IF VI_Sensor_Fault THEN
    L_Sensor_Fault_Clear_Count := 0;
    IF L_Sensor_Fault_Assert_Count < C_HEALTH_DEBOUNCE_CYCLES THEN
        L_Sensor_Fault_Assert_Count := L_Sensor_Fault_Assert_Count + 1;
    END_IF;
    IF L_Sensor_Fault_Assert_Count >= C_HEALTH_DEBOUNCE_CYCLES THEN
        L_Sensor_Fault_Stable := TRUE;
    END_IF;
ELSE
    L_Sensor_Fault_Assert_Count := 0;
    IF L_Sensor_Fault_Clear_Count < C_HEALTH_DEBOUNCE_CYCLES THEN
        L_Sensor_Fault_Clear_Count := L_Sensor_Fault_Clear_Count + 1;
    END_IF;
    IF L_Sensor_Fault_Clear_Count >= C_HEALTH_DEBOUNCE_CYCLES THEN
        L_Sensor_Fault_Stable := FALSE;
    END_IF;
END_IF;

IF VI_Subsystem_Fault THEN
    L_Subsystem_Clear_Count := 0;
    IF L_Subsystem_Assert_Count < C_HEALTH_DEBOUNCE_CYCLES THEN
        L_Subsystem_Assert_Count := L_Subsystem_Assert_Count + 1;
    END_IF;
    IF L_Subsystem_Assert_Count >= C_HEALTH_DEBOUNCE_CYCLES THEN
        L_Subsystem_Fault_Stable := TRUE;
    END_IF;
ELSE
    L_Subsystem_Assert_Count := 0;
    IF L_Subsystem_Clear_Count < C_HEALTH_DEBOUNCE_CYCLES THEN
        L_Subsystem_Clear_Count := L_Subsystem_Clear_Count + 1;
    END_IF;
    IF L_Subsystem_Clear_Count >= C_HEALTH_DEBOUNCE_CYCLES THEN
        L_Subsystem_Fault_Stable := FALSE;
    END_IF;
END_IF;

// Count confirmed fault events on rising edge of stable/critical conditions
IF L_IO_Fault_Stable AND NOT L_IO_Fault_Prev THEN
    VO_IO_Fault_Count := VO_IO_Fault_Count + 1;
END_IF;
L_IO_Fault_Prev := L_IO_Fault_Stable;

IF L_Comm_Fault_Stable AND NOT L_Comm_Fault_Prev THEN
    VO_Comm_Fault_Count := VO_Comm_Fault_Count + 1;
END_IF;
L_Comm_Fault_Prev := L_Comm_Fault_Stable;

IF L_Sensor_Fault_Stable AND NOT L_Sensor_Fault_Prev THEN
    VO_Sensor_Fault_Count := VO_Sensor_Fault_Count + 1;
END_IF;
L_Sensor_Fault_Prev := L_Sensor_Fault_Stable;

IF L_Subsystem_Fault_Stable AND NOT L_Subsystem_Fault_Prev THEN
    VO_Subsystem_Fault_Count := VO_Subsystem_Fault_Count + 1;
END_IF;
L_Subsystem_Fault_Prev := L_Subsystem_Fault_Stable;

IF VI_Watchdog_Fault AND NOT L_Watchdog_Fault_Prev THEN
    VO_Watchdog_Fault_Count := VO_Watchdog_Fault_Count + 1;
END_IF;
L_Watchdog_Fault_Prev := VI_Watchdog_Fault;

VO_Sensor_Fault := L_Sensor_Fault_Stable;
VO_IO_Fault := L_IO_Fault_Stable;
VO_Comm_Fault := L_Comm_Fault_Stable;
VO_Subsystem_Degraded := L_Subsystem_Fault_Stable;

VO_System_Severity := E_System_Severity.SEV_NORMAL;
VO_Root_Cause := E_System_Root_Cause.ROOT_NONE;
VO_First_Fault_Active := FALSE;
VO_First_Fault_Type := 0;
VO_First_Fault_Source := 0;

// Priority: FIRE > GAS > CO > WATER > diagnostics
IF VI_Smoke_Detected THEN
    VO_System_Severity := E_System_Severity.SEV_CRITICAL;
    VO_Root_Cause := E_System_Root_Cause.ROOT_FIRE;
    VO_First_Fault_Active := TRUE;
    VO_First_Fault_Type := 5;

ELSIF VI_Gas_Detected THEN
    VO_System_Severity := E_System_Severity.SEV_CRITICAL;
    VO_Root_Cause := E_System_Root_Cause.ROOT_GAS_LEAK;
    VO_First_Fault_Active := TRUE;
    VO_First_Fault_Type := 6;

ELSIF VI_CO_Alarm_Level THEN
    VO_System_Severity := E_System_Severity.SEV_CRITICAL;
    VO_Root_Cause := E_System_Root_Cause.ROOT_CO_CRITICAL;
    VO_First_Fault_Active := TRUE;
    VO_First_Fault_Type := 7;

ELSIF VI_CO_Warning_Level THEN
    VO_System_Severity := E_System_Severity.SEV_WARNING;
    VO_Root_Cause := E_System_Root_Cause.ROOT_CO_WARNING;
    VO_First_Fault_Active := TRUE;
    VO_First_Fault_Type := 7;

ELSIF VI_Leak_Detected THEN
    VO_System_Severity := E_System_Severity.SEV_WARNING;
    VO_Root_Cause := E_System_Root_Cause.ROOT_WATER_LEAK;
    VO_First_Fault_Active := TRUE;
    VO_First_Fault_Type := 8;

ELSIF VI_Watchdog_Fault THEN
    VO_System_Severity := E_System_Severity.SEV_CRITICAL;
    VO_Root_Cause := E_System_Root_Cause.ROOT_WATCHDOG_FAULT;
    VO_First_Fault_Active := TRUE;
    VO_First_Fault_Type := 9;

ELSIF L_IO_Fault_Stable THEN
    VO_System_Severity := E_System_Severity.SEV_DEGRADED;
    VO_Root_Cause := E_System_Root_Cause.ROOT_IO_OFFLINE;
    VO_First_Fault_Active := TRUE;
    VO_First_Fault_Type := 1;

ELSIF L_Comm_Fault_Stable THEN
    VO_System_Severity := E_System_Severity.SEV_DEGRADED;
    VO_Root_Cause := E_System_Root_Cause.ROOT_COMM_FAULT;
    VO_First_Fault_Active := TRUE;
    VO_First_Fault_Type := 3;

ELSIF L_Sensor_Fault_Stable THEN
    VO_System_Severity := E_System_Severity.SEV_DEGRADED;
    VO_Root_Cause := E_System_Root_Cause.ROOT_SENSOR_FAULT;
    VO_First_Fault_Active := TRUE;
    VO_First_Fault_Type := 2;

ELSIF L_Subsystem_Fault_Stable THEN
    VO_System_Severity := E_System_Severity.SEV_DEGRADED;
    VO_Root_Cause := E_System_Root_Cause.ROOT_SUBSYSTEM_FAULT;
    VO_First_Fault_Active := TRUE;
    VO_First_Fault_Type := 4;
END_IF;
// >>> BULK_SYNC_ANCHOR: FB_System_Health <<<
          
END_FUNCTION_BLOCK

FUNCTION_BLOCK FB_Rule_Engine
  VAR_INPUT
    VI_System_Time_MS : UDINT;
    VI_IsActivePLC : BOOL;
    VI_Security_Armed : BOOL;
    VI_Current_Time : TOD;
    VI_Day_Of_Week : INT;
  END_VAR
  VAR_OUTPUT
    VO_Preheat_Request : BOOL;
    VO_Actions : ARRAY[1..GVL_CONSTANTS.C_MAX_RULES] OF ST_Rule_Action;
  END_VAR
  VAR_IN_OUT
    VI_Rules : ARRAY[1..GVL_CONSTANTS.C_MAX_RULES] OF ST_User_Rule;
    VI_Indoor_Temps : ARRAY[1..16] OF REAL;
    VI_Floor_Temps : ARRAY[1..GVL_CONSTANTS.C_MAX_HEATING_CIRCUITS] OF REAL;
    VI_Humidities : ARRAY[1..16] OF REAL;
    VI_CO2_Levels : ARRAY[1..16] OF REAL;
    VI_Motion_Sensors : ARRAY[1..16] OF BOOL;
    VI_Door_Sensors : ARRAY[1..GVL_CONSTANTS.C_MAX_DOOR_SENSORS] OF BOOL;
    VI_Window_Sensors : ARRAY[1..16] OF BOOL;
    VI_Water_Sensors : ARRAY[1..GVL_CONSTANTS.C_MAX_FLOOD_SENSORS] OF BOOL;
    VI_Smoke_Sensors : ARRAY[1..GVL_CONSTANTS.C_MAX_SMOKE_SENSORS] OF BOOL;
    VI_Methane_Sensors : ARRAY[1..GVL_CONSTANTS.C_MAX_METHANE_SENSORS] OF REAL;
    VI_CO_Sensors : ARRAY[1..GVL_CONSTANTS.C_MAX_CO_SENSORS] OF REAL;
  END_VAR
  VAR
    L_i : INT;
    L_Condition_Met : BOOL;
    L_Current_Value : REAL;
    L_Triggers : ARRAY[1..GVL_CONSTANTS.C_MAX_RULES] OF R_TRIG;
    L_Trigger_Count : ARRAY[1..GVL_CONSTANTS.C_MAX_RULES] OF UINT;
    L_Last_Reset_Time : UDINT;
    L_Elapsed_Time : UDINT;
  END_VAR

            IF NOT VI_IsActivePLC THEN
    FOR L_i := 1 TO GVL_CONSTANTS.C_MAX_RULES DO
        VO_Actions[L_i].Active := FALSE;
        VO_Actions[L_i].Triggered := FALSE;
        VO_Actions[L_i].Action_Type := E_Rule_Action_Type.ACTION_NONE;
        VO_Actions[L_i].Target_ID := 0;
        VO_Actions[L_i].Value := 0.0;
    END_FOR;
    VO_Preheat_Request := FALSE;
    RETURN;
END_IF;

VO_Preheat_Request := FALSE;

L_Elapsed_Time := SEL(VI_System_Time_MS >= L_Last_Reset_Time, VI_System_Time_MS - L_Last_Reset_Time, (4294967295 - L_Last_Reset_Time) + VI_System_Time_MS + 1);

IF L_Elapsed_Time >= GVL_CONSTANTS.C_MS_IN_MINUTE THEN
    L_Last_Reset_Time := VI_System_Time_MS;
    FOR L_i := 1 TO GVL_CONSTANTS.C_MAX_RULES DO
        L_Trigger_Count[L_i] := 0;
    END_FOR;
END_IF;

FOR L_i := 1 TO GVL_CONSTANTS.C_MAX_RULES DO

    // Full per-cycle action reset prevents stale Triggered/Action_Type/Target_ID/Value
    // from being observed by any downstream consumer when a rule is disabled or inactive.
    VO_Actions[L_i].Active := FALSE;
    VO_Actions[L_i].Triggered := FALSE;
    VO_Actions[L_i].Action_Type := E_Rule_Action_Type.ACTION_NONE;
    VO_Actions[L_i].Target_ID := 0;
    VO_Actions[L_i].Value := 0.0;

    IF VI_Rules[L_i].Enabled THEN
        L_Condition_Met := FALSE;
        L_Current_Value := 0.0;
        
        IF VI_Rules[L_i].Condition_Target_ID > 0 THEN
            CASE VI_Rules[L_i].Condition_Type OF
                E_Rule_Condition_Type.COND_AIR_TEMP: IF VI_Rules[L_i].Condition_Target_ID <= 16 THEN L_Current_Value := VI_Indoor_Temps[VI_Rules[L_i].Condition_Target_ID]; END_IF;
                E_Rule_Condition_Type.COND_FLOOR_TEMP: IF VI_Rules[L_i].Condition_Target_ID <= GVL_CONSTANTS.C_MAX_HEATING_CIRCUITS THEN L_Current_Value := VI_Floor_Temps[VI_Rules[L_i].Condition_Target_ID]; END_IF;
                E_Rule_Condition_Type.COND_HUMIDITY: IF VI_Rules[L_i].Condition_Target_ID <= 16 THEN L_Current_Value := VI_Humidities[VI_Rules[L_i].Condition_Target_ID]; END_IF;
                E_Rule_Condition_Type.COND_CO2: IF VI_Rules[L_i].Condition_Target_ID <= 16 THEN L_Current_Value := VI_CO2_Levels[VI_Rules[L_i].Condition_Target_ID]; END_IF;
                E_Rule_Condition_Type.COND_MOTION: IF VI_Rules[L_i].Condition_Target_ID <= 16 THEN L_Current_Value := SEL(VI_Motion_Sensors[VI_Rules[L_i].Condition_Target_ID], 0.0, 1.0); END_IF;
                E_Rule_Condition_Type.COND_DOOR_WINDOW: 
                    IF VI_Rules[L_i].Condition_Target_ID <= GVL_CONSTANTS.C_MAX_DOOR_SENSORS THEN
                        L_Current_Value := SEL(VI_Door_Sensors[VI_Rules[L_i].Condition_Target_ID] OR VI_Window_Sensors[VI_Rules[L_i].Condition_Target_ID], 0.0, 1.0);
                    ELSIF VI_Rules[L_i].Condition_Target_ID <= 16 THEN
                        L_Current_Value := SEL(VI_Window_Sensors[VI_Rules[L_i].Condition_Target_ID], 0.0, 1.0);
                    END_IF;
                E_Rule_Condition_Type.COND_FLOOD: IF VI_Rules[L_i].Condition_Target_ID <= GVL_CONSTANTS.C_MAX_FLOOD_SENSORS THEN L_Current_Value := SEL(VI_Water_Sensors[VI_Rules[L_i].Condition_Target_ID], 0.0, 1.0); END_IF;
                E_Rule_Condition_Type.COND_SMOKE: IF VI_Rules[L_i].Condition_Target_ID <= GVL_CONSTANTS.C_MAX_SMOKE_SENSORS THEN L_Current_Value := SEL(VI_Smoke_Sensors[VI_Rules[L_i].Condition_Target_ID], 0.0, 1.0); END_IF;
                E_Rule_Condition_Type.COND_METHANE: IF VI_Rules[L_i].Condition_Target_ID <= GVL_CONSTANTS.C_MAX_METHANE_SENSORS THEN L_Current_Value := VI_Methane_Sensors[VI_Rules[L_i].Condition_Target_ID]; END_IF;
                E_Rule_Condition_Type.COND_CO: IF VI_Rules[L_i].Condition_Target_ID <= GVL_CONSTANTS.C_MAX_CO_SENSORS THEN L_Current_Value := VI_CO_Sensors[VI_Rules[L_i].Condition_Target_ID]; END_IF;
                E_Rule_Condition_Type.COND_TIME_OF_DAY: L_Current_Value := TO_REAL(TOD_TO_UDINT(VI_Current_Time) / GVL_CONSTANTS.C_MS_IN_MINUTE);
                E_Rule_Condition_Type.COND_DAY_OF_WEEK: L_Current_Value := TO_REAL(VI_Day_Of_Week);
            END_CASE;
        ELSE
            IF VI_Rules[L_i].Condition_Type = E_Rule_Condition_Type.COND_TIME_OF_DAY THEN
                L_Current_Value := TO_REAL(TOD_TO_UDINT(VI_Current_Time) / GVL_CONSTANTS.C_MS_IN_MINUTE);
            ELSIF VI_Rules[L_i].Condition_Type = E_Rule_Condition_Type.COND_DAY_OF_WEEK THEN
                L_Current_Value := TO_REAL(VI_Day_Of_Week);
            END_IF;
        END_IF;
        
        CASE VI_Rules[L_i].Condition_Op OF
            E_Rule_Comparison.COMP_GT: L_Condition_Met := (L_Current_Value > VI_Rules[L_i].Condition_Value);
            E_Rule_Comparison.COMP_LT: L_Condition_Met := (L_Current_Value < VI_Rules[L_i].Condition_Value);
            E_Rule_Comparison.COMP_EQ: L_Condition_Met := (ABS(L_Current_Value - VI_Rules[L_i].Condition_Value) < 0.1);
            E_Rule_Comparison.COMP_GE: L_Condition_Met := (L_Current_Value >= VI_Rules[L_i].Condition_Value);
            E_Rule_Comparison.COMP_LE: L_Condition_Met := (L_Current_Value <= VI_Rules[L_i].Condition_Value);
            E_Rule_Comparison.COMP_IN_RANGE: L_Condition_Met := (L_Current_Value >= VI_Rules[L_i].Condition_Value) AND (L_Current_Value <= VI_Rules[L_i].Condition_Value_Max);
            E_Rule_Comparison.COMP_TRUE: L_Condition_Met := (L_Current_Value > 0.5);
            E_Rule_Comparison.COMP_FALSE: L_Condition_Met := (L_Current_Value < 0.5);
        END_CASE;
        
        L_Triggers[L_i](CLK := L_Condition_Met);
        
        IF L_Triggers[L_i].Q THEN
            L_Trigger_Count[L_i] := L_Trigger_Count[L_i] + 1;
            IF L_Trigger_Count[L_i] > 10 THEN
                CONTINUE;
            END_IF;
        END_IF;
        
        IF L_Condition_Met AND (L_Trigger_Count[L_i] <= 10) THEN
            VO_Actions[L_i].Active := TRUE;
            VO_Actions[L_i].Triggered := L_Triggers[L_i].Q;
            VO_Actions[L_i].Action_Type := VI_Rules[L_i].Action_Type;
            VO_Actions[L_i].Target_ID := VI_Rules[L_i].Action_Target_ID;
            VO_Actions[L_i].Value := VI_Rules[L_i].Action_Value;
        END_IF;
    END_IF;
END_FOR;

// >>> BULK_SYNC_ANCHOR: FB_Rule_Engine <<<
          
END_FUNCTION_BLOCK

FUNCTION_BLOCK FB_Heating_Runtime_Service_Gating_Phase
  VAR_INPUT
    VI_Enable : BOOL;
  END_VAR
  VAR_OUTPUT
    VO_Executed : BOOL;
    VO_Valid : BOOL;
  END_VAR
  VAR_IN_OUT
    VIO_Manifold_Pumps : ARRAY[1..GVL_CONSTANTS.C_MAX_MANIFOLDS] OF BOOL;
    VIO_Backup_Circulation_Pump : BOOL;
    VIO_Electric_Heater_Enable : BOOL;
    VIO_DHW_Heating_Pump : BOOL;
    VIO_DHW_Circ_Pump : BOOL;
    VIO_DHW_Status : ST_DHW_Status;
    VIO_Freeze_Risk_Status : BOOL;
  END_VAR
  VAR
    L_i : INT;
  END_VAR

            // ==============================================================================
// Heating runtime service gating phase
// Applies service/out-of-service and freeze hardware gating to computed outputs.
// Does NOT calculate heating demand and does NOT publish final state.
// ==============================================================================



VO_Executed := FALSE;
VO_Valid := FALSE;

IF NOT VI_Enable THEN
    RETURN;
END_IF;

GVL_STATUS.G_Diagnostics.Backup_Pump_Out_Of_Service := NOT GVL_CONFIG.G_Backup_Circulation_Pump_In_Service;
GVL_STATUS.G_Diagnostics.Electric_Heater_Out_Of_Service := NOT GVL_CONFIG.G_Electric_Heater_In_Service;

IF NOT GVL_CONFIG.G_Backup_Circulation_Pump_In_Service THEN
    VIO_Backup_Circulation_Pump := FALSE;
END_IF;

IF NOT GVL_CONFIG.G_Electric_Heater_In_Service THEN
    VIO_Electric_Heater_Enable := FALSE;
END_IF;

FOR L_i := 1 TO GVL_CONSTANTS.C_MAX_MANIFOLDS DO
    GVL_STATUS.G_Diagnostics.Manifold_Pump_Out_Of_Service[L_i] := NOT GVL_CONFIG.G_Manifold_Pump_In_Service[L_i];
    IF NOT GVL_CONFIG.G_Manifold_Pump_In_Service[L_i] THEN
        VIO_Manifold_Pumps[L_i] := FALSE;
    END_IF;
END_FOR;

GVL_STATUS.G_Diagnostics.DHW_Heating_Pump_Out_Of_Service := NOT GVL_CONFIG.G_DHW_Heating_Pump_In_Service;
IF NOT GVL_CONFIG.G_DHW_Heating_Pump_In_Service THEN
    VIO_DHW_Heating_Pump := FALSE;
    VIO_DHW_Status.Heating_Pump_On := FALSE;
END_IF;

GVL_STATUS.G_Diagnostics.DHW_Circ_Pump_Out_Of_Service := NOT GVL_CONFIG.G_DHW_Circ_Pump_In_Service;
IF NOT GVL_CONFIG.G_DHW_Circ_Pump_In_Service THEN
    VIO_DHW_Circ_Pump := FALSE;
    VIO_DHW_Status.Circ_Pump_On := FALSE;
END_IF;

GVL_STATE.G_Freeze_Hardware_Degraded := GVL_STATUS.G_Diagnostics.Backup_Pump_Fault OR GVL_STATUS.G_Diagnostics.Electric_Heater_Fault;
GVL_STATE.G_Freeze_Hardware_Failed := GVL_STATUS.G_Diagnostics.Backup_Pump_Fault AND GVL_STATUS.G_Diagnostics.Electric_Heater_Fault;

IF GVL_STATE.G_Freeze_Hardware_Failed THEN
    VIO_Backup_Circulation_Pump := FALSE;
    VIO_Electric_Heater_Enable := FALSE;
    VIO_Freeze_Risk_Status := TRUE;
END_IF;

VO_Executed := TRUE;
VO_Valid := TRUE;

// >>> BULK_SYNC_ANCHOR: FB_Heating_Runtime_Service_Gating_Phase <<<
          
END_FUNCTION_BLOCK

FUNCTION_BLOCK FB_OPCUA_Runtime_Adapter
  VAR_INPUT
    VI_Enable : BOOL;
    VI_System_Time_MS : UDINT;
  END_VAR
  VAR
    L_Frame : ST_Runtime_Bus_Frame;
    L_TX_Index : UINT;
  END_VAR

            IF NOT VI_Enable THEN
    RETURN;
END_IF;

L_TX_Index := UDINT_TO_UINT(GVL_Runtime_Bus.G_Last_Sequence_Id);

IF (L_TX_Index >= 1)
   AND (L_TX_Index <= 128) THEN

    L_Frame := GVL_Runtime_Bus.G_TX_Frames[L_TX_Index];

    IF L_Frame.Frame_Valid THEN

        IF GVL_Distributed_Authority.G_Distributed_Safety_Barrier_OK
           AND NOT GVL_Runtime_Discovery.G_Any_Node_Quarantined THEN

            L_Frame.Frame_Ack_Received := TRUE;
            L_Frame.Replication_Consistent := TRUE;
            L_Frame.Status_Code := 0;

        ELSE

            L_Frame.Replication_Rejected := TRUE;
            L_Frame.Status_Code := 2;

        END_IF;

        GVL_Runtime_Bus.G_TX_Frames[L_TX_Index] := L_Frame;

    END_IF;

END_IF;
          
END_FUNCTION_BLOCK

FUNCTION_BLOCK FB_Modbus_RTU_SysCom_Backend
  VAR_INPUT
    VI_Enable : BOOL;
    VI_System_Time_MS : UDINT;
  END_VAR
  VAR
    L_Result : UDINT;
    L_Handle : UDINT := 16#FFFFFFFF;
    L_Settings : SysCom.SysComSettings;
    L_SettingsEx2 : SysCom.SysComSettingsEx2;
    L_Bytes_Written : UDINT;
    L_Bytes_Read : UDINT;
    L_RX_Buffer : ARRAY[0..255] OF BYTE;
    L_Open_Done : BOOL := FALSE;
    L_i : INT;
    L_j : INT;
    L_Read_Count : INT;
    L_Target_Index : INT;
    L_Frame_Length : INT;
    L_CRC : WORD;
    L_CRC_Frame : WORD;
    L_Baudrate : UDINT;
    L_Interframe_MS : UDINT;
  END_VAR

            // ======================================================
// MODBUS RTU SYSCOM BACKEND
// ======================================================
// Industrial transport runtime:
//   - serial open/configure
//   - RX assembler
//   - CRC validation
//   - watchdog supervision
//   - reconnect supervision
// ======================================================

IF NOT VI_Enable THEN

    IF L_Handle <> 16#FFFFFFFF THEN
        SysCom.SysComClose(hCom := L_Handle);
        L_Handle := 16#FFFFFFFF;
    END_IF;

    L_Open_Done := FALSE;

    GVL_MODBUS_SYSCOM_TRANSPORT.G_Transport_Attached := FALSE;
    GVL_MODBUS_SYSCOM_TRANSPORT.G_Backend_Online := FALSE;

    GVL_MODBUS_SYSCOM_TRANSPORT.G_Backend_State :=
        MB_SYSCOM_CLOSED;

    GVL_MODBUS_SYSCOM_TRANSPORT.G_RX_State :=
        MB_RTU_RX_IDLE;

    GVL_MODBUS_SYSCOM_TRANSPORT.G_RX_Assembler_Active := FALSE;
    GVL_MODBUS_SYSCOM_TRANSPORT.G_RX_Assembler_Length := 0;

    RETURN;
END_IF;

// ======================================================
// WATCHDOGS
// ======================================================
GVL_MODBUS_SYSCOM_TRANSPORT.G_TX_Watchdog_Timeout := FALSE;
GVL_MODBUS_SYSCOM_TRANSPORT.G_RX_Watchdog_Timeout := FALSE;
GVL_MODBUS_SYSCOM_TRANSPORT.G_Bus_Silent := FALSE;

IF GVL_MODBUS_SYSCOM_TRANSPORT.G_TX_Request THEN

    IF (VI_System_Time_MS -
        GVL_MODBUS_SYSCOM_TRANSPORT.G_Last_TX_Request_MS) >
        (GVL_CONFIG.G_Modbus_RTU_Request_Timeout_MS * 2) THEN

        GVL_MODBUS_SYSCOM_TRANSPORT.G_TX_Watchdog_Timeout := TRUE;

        GVL_MODBUS_SYSCOM_TRANSPORT.G_Total_TX_Watchdog :=
            GVL_MODBUS_SYSCOM_TRANSPORT.G_Total_TX_Watchdog + 1;

    END_IF;

END_IF;

IF GVL_MODBUS_SYSCOM_TRANSPORT.G_Backend_Online THEN

    IF (VI_System_Time_MS -
        GVL_MODBUS_SYSCOM_TRANSPORT.G_Last_RX_MS) > 30000 THEN

        GVL_MODBUS_SYSCOM_TRANSPORT.G_RX_Watchdog_Timeout := TRUE;

        GVL_MODBUS_SYSCOM_TRANSPORT.G_Total_RX_Watchdog :=
            GVL_MODBUS_SYSCOM_TRANSPORT.G_Total_RX_Watchdog + 1;

        GVL_MODBUS_SYSCOM_TRANSPORT.G_Bus_Silent := TRUE;

    END_IF;

END_IF;

// ======================================================
// RECONNECT WAIT STATE
// ======================================================
IF GVL_MODBUS_SYSCOM_TRANSPORT.G_Backend_State =
   MB_SYSCOM_RECONNECT_WAIT THEN

    IF (VI_System_Time_MS -
        GVL_MODBUS_SYSCOM_TRANSPORT.G_Backend_Last_Error_MS) >=
        GVL_MODBUS_SYSCOM_TRANSPORT.G_Backend_Reconnect_Delay_MS THEN

        GVL_MODBUS_SYSCOM_TRANSPORT.G_Backend_State :=
            MB_SYSCOM_OPENING;

    ELSE

        RETURN;

    END_IF;

END_IF;

// ======================================================
// OPEN + CONFIGURE
// ======================================================
IF NOT L_Open_Done THEN

    GVL_MODBUS_SYSCOM_TRANSPORT.G_Backend_State :=
        MB_SYSCOM_OPENING;

    L_Baudrate := GVL_CONFIG.G_Modbus_RTU_Baudrate;

    IF L_Baudrate <= 9600 THEN
        L_Interframe_MS := 5;
    ELSIF L_Baudrate <= 19200 THEN
        L_Interframe_MS := 3;
    ELSE
        L_Interframe_MS := 2;
    END_IF;

    GVL_MODBUS_SYSCOM_TRANSPORT.G_RX_Assembler_InterFrame_MS :=
        L_Interframe_MS;

    CASE GVL_CONFIG.G_Modbus_RTU_Port_Number OF
        1:
            L_Settings.sPort := SysCom.SYS_COMPORT1;
        2:
            L_Settings.sPort := SysCom.SYS_COMPORT2;
        3:
            L_Settings.sPort := SysCom.SYS_COMPORT3;
        4:
            L_Settings.sPort := SysCom.SYS_COMPORT4;
    ELSE
        L_Settings.sPort := SysCom.SYS_COMPORT1;
    END_CASE;

    CASE GVL_CONFIG.G_Modbus_RTU_Baudrate OF
        4800:
            L_Settings.ulBaudrate := SysCom.SYS_BR_4800;
        9600:
            L_Settings.ulBaudrate := SysCom.SYS_BR_9600;
        19200:
            L_Settings.ulBaudrate := SysCom.SYS_BR_19200;
        38400:
            L_Settings.ulBaudrate := SysCom.SYS_BR_38400;
        57600:
            L_Settings.ulBaudrate := SysCom.SYS_BR_57600;
        115200:
            L_Settings.ulBaudrate := SysCom.SYS_BR_115200;
    ELSE
        L_Settings.ulBaudrate := SysCom.SYS_BR_9600;
    END_CASE;

    CASE GVL_CONFIG.G_Modbus_RTU_Parity OF
        0:
            L_Settings.byParity := SysCom.SYS_NOPARITY;
        1:
            L_Settings.byParity := SysCom.SYS_EVENPARITY;
        2:
            L_Settings.byParity := SysCom.SYS_ODDPARITY;
    ELSE
        L_Settings.byParity := SysCom.SYS_EVENPARITY;
    END_CASE;

    CASE GVL_CONFIG.G_Modbus_RTU_Stop_Bits OF
        1:
            L_Settings.byStopBits := SysCom.SYS_ONESTOPBIT;
        2:
            L_Settings.byStopBits := SysCom.SYS_TWOSTOPBITS;
    ELSE
        L_Settings.byStopBits := SysCom.SYS_ONESTOPBIT;
    END_CASE;

    L_Settings.ulTimeout := GVL_CONFIG.G_Modbus_RTU_Request_Timeout_MS;
    L_Settings.ulBufferSize := 512;

    IF GVL_CONFIG.G_Modbus_RTU_Data_Bits < 7 THEN
        L_SettingsEx2.byByteSize := 8;
    ELSIF GVL_CONFIG.G_Modbus_RTU_Data_Bits > 8 THEN
        L_SettingsEx2.byByteSize := 8;
    ELSE
        L_SettingsEx2.byByteSize := GVL_CONFIG.G_Modbus_RTU_Data_Bits;
    END_IF;

    L_SettingsEx2.bBinary := TRUE;
    L_SettingsEx2.bOutxCtsFlow := FALSE;
    L_SettingsEx2.bOutxDsrFlow := FALSE;
    L_SettingsEx2.byDtrControl := 0;
    L_SettingsEx2.bDsrSensitivity := FALSE;
    L_SettingsEx2.byRtsControl := 0;
    L_SettingsEx2.bTXContinueOnXoff := FALSE;
    L_SettingsEx2.bOutX := FALSE;
    L_SettingsEx2.bInX := FALSE;
    L_SettingsEx2.byXonChar := 0;
    L_SettingsEx2.byXoffChar := 0;
    L_SettingsEx2.wXonLim := 0;
    L_SettingsEx2.wXoffLim := 0;

    L_Handle := SysCom.SysComOpen3(
        pSettings := ADR(L_Settings),
        pSettingsEx2 := ADR(L_SettingsEx2),
        pResult := ADR(L_Result)
    );

    IF L_Handle <> 16#FFFFFFFF THEN

        SysCom.SysComPurge(hCom := L_Handle);

        L_Open_Done := TRUE;

        GVL_MODBUS_SYSCOM_TRANSPORT.G_Transport_Attached := TRUE;
        GVL_MODBUS_SYSCOM_TRANSPORT.G_Backend_Online := TRUE;

        GVL_MODBUS_SYSCOM_TRANSPORT.G_Backend_State :=
            MB_SYSCOM_ONLINE;

    ELSE

        GVL_MODBUS_SYSCOM_TRANSPORT.G_Transport_Attached := FALSE;
        GVL_MODBUS_SYSCOM_TRANSPORT.G_Backend_Online := FALSE;

        GVL_MODBUS_SYSCOM_TRANSPORT.G_Backend_State :=
            MB_SYSCOM_RECONNECT_WAIT;

        GVL_MODBUS_SYSCOM_TRANSPORT.G_Backend_Last_Error_MS :=
            VI_System_Time_MS;

        GVL_MODBUS_SYSCOM_TRANSPORT.G_Backend_Reconnect_Attempts :=
            GVL_MODBUS_SYSCOM_TRANSPORT.G_Backend_Reconnect_Attempts + 1;

        GVL_MODBUS_SYSCOM_TRANSPORT.G_Total_Reconnects :=
            GVL_MODBUS_SYSCOM_TRANSPORT.G_Total_Reconnects + 1;

        GVL_MODBUS_SYSCOM_TRANSPORT.G_Total_Errors :=
            GVL_MODBUS_SYSCOM_TRANSPORT.G_Total_Errors + 1;

    END_IF;

    RETURN;
END_IF;

GVL_MODBUS_SYSCOM_TRANSPORT.G_Backend_State :=
    MB_SYSCOM_ONLINE;

// ======================================================
// TX WRITE
// ======================================================
IF GVL_MODBUS_SYSCOM_TRANSPORT.G_TX_Request AND
   NOT GVL_MODBUS_SYSCOM_TRANSPORT.G_TX_Done THEN

    L_Bytes_Written := SysCom.SysComWrite(
        hCom := L_Handle,
        pbyBuffer := ADR(GVL_MODBUS_SYSCOM_TRANSPORT.G_TX_Buffer),
        ulSize := GVL_MODBUS_SYSCOM_TRANSPORT.G_TX_Length,
        ulTimeout := GVL_CONFIG.G_Modbus_RTU_Request_Timeout_MS,
        pResult := ADR(L_Result)
    );

    IF L_Bytes_Written = GVL_MODBUS_SYSCOM_TRANSPORT.G_TX_Length THEN

        GVL_MODBUS_SYSCOM_TRANSPORT.G_TX_Done := TRUE;

    ELSE

        GVL_MODBUS_SYSCOM_TRANSPORT.G_TX_Error := TRUE;

        GVL_MODBUS_SYSCOM_TRANSPORT.G_Backend_State :=
            MB_SYSCOM_ERROR;

    END_IF;

END_IF;

// ======================================================
// RX STREAM READ
// ======================================================
L_Bytes_Read := SysCom.SysComRead(
    hCom := L_Handle,
    pbyBuffer := ADR(L_RX_Buffer),
    ulSize := 256,
    ulTimeout := SysCom.SYS_NOWAIT,
    pResult := ADR(L_Result)
);

IF L_Bytes_Read > 0 THEN

    GVL_MODBUS_SYSCOM_TRANSPORT.G_RX_State :=
        MB_RTU_RX_RECEIVING;

    IF L_Bytes_Read > 256 THEN
        L_Read_Count := 256;
    ELSE
        L_Read_Count := UDINT_TO_INT(L_Bytes_Read);
    END_IF;

    GVL_MODBUS_SYSCOM_TRANSPORT.G_RX_Assembler_Active := TRUE;

    GVL_MODBUS_SYSCOM_TRANSPORT.G_RX_Assembler_Last_Byte_MS :=
        VI_System_Time_MS;

    FOR L_i := 0 TO (L_Read_Count - 1) DO

        L_Target_Index :=
            UINT_TO_INT(GVL_MODBUS_SYSCOM_TRANSPORT.G_RX_Assembler_Length);

        IF L_Target_Index >= 256 THEN

            GVL_MODBUS_SYSCOM_TRANSPORT.G_RX_State :=
                MB_RTU_RX_OVERFLOW;

            GVL_MODBUS_SYSCOM_TRANSPORT.G_RX_Assembler_Overflow := TRUE;

            GVL_MODBUS_SYSCOM_TRANSPORT.G_Total_RX_Overflow :=
                GVL_MODBUS_SYSCOM_TRANSPORT.G_Total_RX_Overflow + 1;

            GVL_MODBUS_SYSCOM_TRANSPORT.G_RX_Assembler_Active := FALSE;
            GVL_MODBUS_SYSCOM_TRANSPORT.G_RX_Assembler_Length := 0;

            EXIT;

        END_IF;

        GVL_MODBUS_SYSCOM_TRANSPORT.G_RX_Buffer[L_Target_Index] :=
            L_RX_Buffer[L_i];

        GVL_MODBUS_SYSCOM_TRANSPORT.G_RX_Assembler_Length :=
            GVL_MODBUS_SYSCOM_TRANSPORT.G_RX_Assembler_Length + 1;

    END_FOR;

END_IF;

// ======================================================
// INTER-FRAME FINALIZATION
// ======================================================
IF GVL_MODBUS_SYSCOM_TRANSPORT.G_RX_Assembler_Active THEN

    IF (VI_System_Time_MS -
        GVL_MODBUS_SYSCOM_TRANSPORT.G_RX_Assembler_Last_Byte_MS) >=
        GVL_MODBUS_SYSCOM_TRANSPORT.G_RX_Assembler_InterFrame_MS THEN

        L_Frame_Length :=
            UINT_TO_INT(GVL_MODBUS_SYSCOM_TRANSPORT.G_RX_Assembler_Length);

        IF L_Frame_Length >= 4 THEN

            L_CRC := 16#FFFF;

            FOR L_i := 0 TO (L_Frame_Length - 3) DO

                L_CRC := L_CRC XOR
                    BYTE_TO_WORD(
                        GVL_MODBUS_SYSCOM_TRANSPORT.G_RX_Buffer[L_i]
                    );

                FOR L_j := 0 TO 7 DO

                    IF (L_CRC AND 16#0001) <> 0 THEN
                        L_CRC := SHR(L_CRC, 1);
                        L_CRC := L_CRC XOR 16#A001;
                    ELSE
                        L_CRC := SHR(L_CRC, 1);
                    END_IF;

                END_FOR;

            END_FOR;

            L_CRC_Frame :=
                BYTE_TO_WORD(
                    GVL_MODBUS_SYSCOM_TRANSPORT.G_RX_Buffer[L_Frame_Length - 2]
                );

            L_CRC_Frame :=
                L_CRC_Frame OR
                SHL(
                    BYTE_TO_WORD(
                        GVL_MODBUS_SYSCOM_TRANSPORT.G_RX_Buffer[L_Frame_Length - 1]
                    ),
                    8
                );

            GVL_MODBUS_SYSCOM_TRANSPORT.G_RX_Assembler_CRC_Calc :=
                L_CRC;

            GVL_MODBUS_SYSCOM_TRANSPORT.G_RX_Assembler_CRC_Frame :=
                L_CRC_Frame;

            IF L_CRC = L_CRC_Frame THEN

                GVL_MODBUS_SYSCOM_TRANSPORT.G_RX_State :=
                    MB_RTU_RX_FRAME_READY;

                GVL_MODBUS_SYSCOM_TRANSPORT.G_RX_Assembler_CRC_OK := TRUE;

                GVL_MODBUS_SYSCOM_TRANSPORT.G_RX_Length :=
                    GVL_MODBUS_SYSCOM_TRANSPORT.G_RX_Assembler_Length;

                GVL_MODBUS_SYSCOM_TRANSPORT.G_RX_Ready := TRUE;

                GVL_MODBUS_SYSCOM_TRANSPORT.G_Total_RX :=
                    GVL_MODBUS_SYSCOM_TRANSPORT.G_Total_RX + 1;

                GVL_MODBUS_SYSCOM_TRANSPORT.G_Last_RX_MS :=
                    VI_System_Time_MS;

            ELSE

                GVL_MODBUS_SYSCOM_TRANSPORT.G_RX_State :=
                    MB_RTU_RX_CRC_ERROR;

                GVL_MODBUS_SYSCOM_TRANSPORT.G_RX_Assembler_CRC_OK := FALSE;

                GVL_MODBUS_SYSCOM_TRANSPORT.G_Total_RX_CRC_Error :=
                    GVL_MODBUS_SYSCOM_TRANSPORT.G_Total_RX_CRC_Error + 1;

            END_IF;

        ELSE

            GVL_MODBUS_SYSCOM_TRANSPORT.G_RX_State :=
                MB_RTU_RX_SHORT_FRAME;

            GVL_MODBUS_SYSCOM_TRANSPORT.G_Total_RX_Short_Frame :=
                GVL_MODBUS_SYSCOM_TRANSPORT.G_Total_RX_Short_Frame + 1;

        END_IF;

        GVL_MODBUS_SYSCOM_TRANSPORT.G_RX_Assembler_Active := FALSE;
        GVL_MODBUS_SYSCOM_TRANSPORT.G_RX_Assembler_Length := 0;

    END_IF;

END_IF;

IF NOT GVL_MODBUS_SYSCOM_TRANSPORT.G_RX_Assembler_Active AND
   NOT GVL_MODBUS_SYSCOM_TRANSPORT.G_RX_Ready AND
   (GVL_MODBUS_SYSCOM_TRANSPORT.G_RX_State = MB_RTU_RX_FRAME_READY) THEN

    GVL_MODBUS_SYSCOM_TRANSPORT.G_RX_State :=
        MB_RTU_RX_IDLE;

END_IF;
          
END_FUNCTION_BLOCK

FUNCTION_BLOCK FB_Modbus_Response_Apply
  VAR_INPUT
    VI_Request_Valid : BOOL;
    VI_Request_Index : INT;
    VI_Request_Sequence : UDINT;
    VI_Parser_Valid : BOOL;
    VI_Parser_Error : BOOL;
    VI_Parser_Error_Code : WORD;
    VI_Register_Count : UINT;
    VI_Register_Value : ARRAY[1..32] OF WORD;
    VI_System_Time_MS : UDINT;
  END_VAR
  VAR_OUTPUT
    VO_Response_Applied : BOOL;
  END_VAR
  VAR
    L_i : INT;
    L_Count : INT;
  END_VAR

            // ======================================================
// MODBUS RESPONSE APPLY LAYER
// ======================================================
// Transfers validated parser result into bridge/master response.
//
// Safety principles:
//   - Only validated parser result may produce Done.
//   - Parser error produces Error response.
//   - No synthetic successful response.
// ======================================================

VO_Response_Applied := FALSE;

IF NOT VI_Request_Valid THEN
    RETURN;
END_IF;

IF (VI_Request_Index < 1) OR (VI_Request_Index > 16) THEN
    RETURN;
END_IF;

// ======================================================
// PARSER ERROR
// ======================================================
IF VI_Parser_Error THEN

    GVL_MODBUS_RTU_BRIDGE.G_Response_Busy := FALSE;
    GVL_MODBUS_RTU_BRIDGE.G_Response_Done := FALSE;
    GVL_MODBUS_RTU_BRIDGE.G_Response_Error := TRUE;
    GVL_MODBUS_RTU_BRIDGE.G_Response_Error_Code := VI_Parser_Error_Code;
    GVL_MODBUS_RTU_BRIDGE.G_Response_Sequence := VI_Request_Sequence;
    GVL_MODBUS_RTU_BRIDGE.G_Response_Update_MS := VI_System_Time_MS;

    VO_Response_Applied := TRUE;

    RETURN;
END_IF;

// ======================================================
// VALID PARSED RESPONSE
// ======================================================
IF VI_Parser_Valid THEN

    FOR L_i := 1 TO 32 DO
        GVL_MODBUS_RTU_BRIDGE.G_Response_Value[L_i] := 0;
    END_FOR;

    L_Count := UINT_TO_INT(VI_Register_Count);

    IF L_Count > 32 THEN
        L_Count := 32;
    END_IF;

    FOR L_i := 1 TO L_Count DO
        GVL_MODBUS_RTU_BRIDGE.G_Response_Value[L_i] :=
            VI_Register_Value[L_i];
    END_FOR;

    GVL_MODBUS_RTU_BRIDGE.G_Response_Busy := FALSE;
    GVL_MODBUS_RTU_BRIDGE.G_Response_Done := TRUE;
    GVL_MODBUS_RTU_BRIDGE.G_Response_Error := FALSE;
    GVL_MODBUS_RTU_BRIDGE.G_Response_Error_Code := 0;
    GVL_MODBUS_RTU_BRIDGE.G_Response_Sequence := VI_Request_Sequence;
    GVL_MODBUS_RTU_BRIDGE.G_Response_Update_MS := VI_System_Time_MS;

    VO_Response_Applied := TRUE;

END_IF;
          
END_FUNCTION_BLOCK

FUNCTION_BLOCK FB_Heating_Safe_State
  VAR_INPUT
    VI_Block_Normal_Heating : BOOL;
    VI_IO_Failsafe_Active : BOOL;
    VI_Gas_Safety_Active : BOOL;
    VI_Freeze_Active : BOOL;
    VI_Freeze_Target_Supply : REAL;
    VI_Manifold_Temps_Supply : ARRAY[1..GVL_CONSTANTS.C_MAX_MANIFOLDS] OF REAL;
    VI_Boiler_Error_Status : ARRAY[1..GVL_CONSTANTS.C_MAX_BOILERS] OF BOOL;
    VI_Boiler_OT_Online : ARRAY[1..GVL_CONSTANTS.C_MAX_BOILERS] OF BOOL;
  END_VAR
  VAR_OUTPUT
    VO_Applied : BOOL;
    VO_Zone_Valves : ARRAY[1..GVL_CONSTANTS.C_MAX_HEATING_CIRCUITS] OF BOOL;
    VO_Manifold_Pumps : ARRAY[1..GVL_CONSTANTS.C_MAX_MANIFOLDS] OF BOOL;
    VO_Manifold_Valves : ARRAY[1..GVL_CONSTANTS.C_MAX_MANIFOLDS] OF REAL;
    VO_Boiler_OT_Enable : ARRAY[1..GVL_CONSTANTS.C_MAX_BOILERS] OF BOOL;
    VO_Boiler_OT_Setpoint : ARRAY[1..GVL_CONSTANTS.C_MAX_BOILERS] OF REAL;
    VO_Boiler_Status : ARRAY[1..GVL_CONSTANTS.C_MAX_BOILERS] OF ST_Boiler_Status;
    VO_Backup_Circulation_Pump : BOOL;
    VO_Electric_Heater_Enable : BOOL;
    VO_Freeze_Risk_Status : BOOL;
  END_VAR
  VAR
    L_i : INT;
    L_Min_Supply_Temp : REAL;
    L_Freeze_Circulation_Required : BOOL;
  END_VAR

            VO_Applied := VI_Block_Normal_Heating;
VO_Backup_Circulation_Pump := FALSE;
VO_Electric_Heater_Enable := FALSE;
VO_Freeze_Risk_Status := FALSE;

L_Freeze_Circulation_Required := VI_Freeze_Active AND (VI_IO_Failsafe_Active OR VI_Gas_Safety_Active);

IF NOT VI_Block_Normal_Heating THEN
    RETURN;
END_IF;

// =============================
// ZONE VALVES (FIXED)
// =============================
FOR L_i := 1 TO GVL_CONSTANTS.C_MAX_HEATING_CIRCUITS DO
    IF L_Freeze_Circulation_Required THEN
        VO_Zone_Valves[L_i] := TRUE;
    ELSE
        VO_Zone_Valves[L_i] := FALSE;
    END_IF;
END_FOR;

// =============================
// MANIFOLD CONTROL
// =============================
FOR L_i := 1 TO GVL_CONSTANTS.C_MAX_MANIFOLDS DO
    IF L_Freeze_Circulation_Required THEN
        VO_Manifold_Pumps[L_i] := TRUE;
        VO_Manifold_Valves[L_i] := REAL#35.0;
    ELSE
        VO_Manifold_Pumps[L_i] := FALSE;
        VO_Manifold_Valves[L_i] := REAL#0.0;
    END_IF;
END_FOR;

// =============================
// BOILERS OFF
// =============================
FOR L_i := 1 TO GVL_CONSTANTS.C_MAX_BOILERS DO
    VO_Boiler_OT_Enable[L_i] := FALSE;
    VO_Boiler_OT_Setpoint[L_i] := REAL#0.0;
    VO_Boiler_Status[L_i].Warning := FALSE;
    VO_Boiler_Status[L_i].Error := TRUE;
END_FOR;

// =============================
// FREEZE PROTECTION LOGIC
// =============================
IF VI_Gas_Safety_Active AND VI_Freeze_Active THEN
    VO_Backup_Circulation_Pump := TRUE;

    L_Min_Supply_Temp := REAL#1000.0;
    FOR L_i := 1 TO GVL_CONSTANTS.C_MAX_MANIFOLDS DO
        IF VI_Manifold_Temps_Supply[L_i] < L_Min_Supply_Temp THEN
            L_Min_Supply_Temp := VI_Manifold_Temps_Supply[L_i];
        END_IF;
    END_FOR;

    IF L_Min_Supply_Temp > REAL#900.0 THEN
        L_Min_Supply_Temp := REAL#0.0;
    END_IF;

    IF L_Min_Supply_Temp < (VI_Freeze_Target_Supply - REAL#1.0) THEN
        VO_Electric_Heater_Enable := TRUE;
    ELSIF L_Min_Supply_Temp > (VI_Freeze_Target_Supply + REAL#1.0) THEN
        VO_Electric_Heater_Enable := FALSE;
    END_IF;

    VO_Freeze_Risk_Status := TRUE;
END_IF;

// =============================
// IO FAILSAFE + FREEZE
// =============================
IF VI_IO_Failsafe_Active AND VI_Freeze_Active THEN
    IF VI_Boiler_OT_Online[1] AND NOT VI_Boiler_Error_Status[1] THEN
        VO_Boiler_OT_Enable[1] := TRUE;
        VO_Boiler_OT_Setpoint[1] := VI_Freeze_Target_Supply;
    END_IF;
END_IF;

// >>> BULK_SYNC_ANCHOR: FB_Heating_Safe_State <<<
          
END_FUNCTION_BLOCK

FUNCTION_BLOCK FB_Heating_Runtime_RootCause_Correlator
  VAR_INPUT
    VI_Enable : BOOL;
    VI_Anomaly : ST_Heating_Runtime_Anomaly;
  END_VAR
  VAR_OUTPUT
    VO_Node : ST_Heating_Runtime_Causality_Node;
  END_VAR

            // ==============================================================================
// Heating runtime root-cause correlator
// Read-only runtime causality correlation layer.
// ==============================================================================



VO_Node.Node_Active := FALSE;
VO_Node.Root_Cause_Candidate := FALSE;
VO_Node.Runtime_Degraded := FALSE;
VO_Node.Runtime_Fault := FALSE;

VO_Node.Cascade_Degraded := FALSE;
VO_Node.Cascade_Boiler_Loss := FALSE;

VO_Node.OpenTherm_Degraded := FALSE;
VO_Node.OpenTherm_Command_Invalid := FALSE;

VO_Node.Diagnostics_Degraded := FALSE;
VO_Node.Explainability_Degraded := FALSE;

VO_Node.Sequencing_Invalid := FALSE;
VO_Node.Ownership_Invalid := FALSE;
VO_Node.Synchronization_Invalid := FALSE;

VO_Node.Severity_Level := 0;

VO_Node.Status_Code := 0;
VO_Node.Status_Text := 'Heating runtime root-cause correlator disabled';

IF NOT VI_Enable THEN
    RETURN;
END_IF;

VO_Node.Node_Active := VI_Anomaly.Anomaly_Active;

VO_Node.Runtime_Degraded := VI_Anomaly.Runtime_Degraded;
VO_Node.Runtime_Fault :=
    VI_Anomaly.Critical_Anomaly;

VO_Node.Cascade_Degraded :=
    VI_Anomaly.Cascade_Degraded;

VO_Node.Cascade_Boiler_Loss :=
    VI_Anomaly.Cascade_Boiler_Loss_Detected;

VO_Node.OpenTherm_Degraded :=
    VI_Anomaly.OpenTherm_Transport_Degraded;

VO_Node.OpenTherm_Command_Invalid :=
    VI_Anomaly.OpenTherm_Command_Invalid;

VO_Node.Diagnostics_Degraded :=
    VI_Anomaly.Diagnostics_Degraded;

VO_Node.Explainability_Degraded :=
    VI_Anomaly.Explainability_Degraded;

VO_Node.Sequencing_Invalid :=
    VI_Anomaly.Sequencing_Invalid;

VO_Node.Ownership_Invalid :=
    VI_Anomaly.Ownership_Invalid;

VO_Node.Synchronization_Invalid :=
    VI_Anomaly.Synchronization_Invalid;

VO_Node.Severity_Level :=
    VI_Anomaly.Severity_Level;

VO_Node.Root_Cause_Candidate :=
    VI_Anomaly.Critical_Anomaly OR
    VI_Anomaly.Sequencing_Invalid OR
    VI_Anomaly.Ownership_Invalid OR
    VI_Anomaly.Synchronization_Invalid;

IF VO_Node.Root_Cause_Candidate THEN
    VO_Node.Status_Code := 900;
    VO_Node.Status_Text := 'Heating runtime root-cause candidate detected';
ELSE
    VO_Node.Status_Code := 1;
    VO_Node.Status_Text := 'Heating runtime causality nominal';
END_IF;

// >>> BULK_SYNC_ANCHOR: FB_Heating_Runtime_RootCause_Correlator <<<
          
END_FUNCTION_BLOCK

FUNCTION_BLOCK FB_System_Init
  VAR_IN_OUT
    VIO_Local_State : ST_System_State_Snapshot;
    VIO_Remote_State : ST_System_State_Snapshot;
  END_VAR
  VAR
    L_i : INT;
  END_VAR

            // ==============================================================================
// System init helper
//
// Internal helper for PRG_System.
// Owns first-boot initialization of RETAIN runtime state.
// ==============================================================================



IF NOT GVL_Retain.G_Initialized THEN
    FOR L_i := 0 TO GVL_CONSTANTS.C_MAX_PRESENCE_HISTORY - 1 DO
        GVL_Retain.G_Presence_History[L_i] := 0;
    END_FOR;

    GVL_Retain.G_History_Write_Idx := 1;
    GVL_Retain.G_History_Total_Events := 0;

    FOR L_i := 1 TO GVL_CONSTANTS.C_MAX_BOILERS DO
        GVL_Retain.G_Boiler_Accumulated_MS[L_i] := 0;
        GVL_Retain.G_Boiler_Work_Seconds[L_i] := 0;
    END_FOR;

    FOR L_i := 1 TO GVL_CONSTANTS.C_MAX_MANIFOLDS DO
        GVL_Retain.G_Valve_Test_Results[L_i] := FALSE;
    END_FOR;

    VIO_Local_State.Version := 0;
    VIO_Remote_State.Version := 0;

    GVL_Retain.G_Initialized := TRUE;
END_IF;

// >>> BULK_SYNC_ANCHOR: FB_System_Init <<<
          
END_FUNCTION_BLOCK

FUNCTION_BLOCK FB_Analog_Validator
  VAR_INPUT
    VI_Value : REAL;
    VI_Min_Valid : REAL;
    VI_Max_Valid : REAL;
    VI_Fallback_Mode : INT := 0;
    VI_Default_Value : REAL := 0.0;
  END_VAR
  VAR_OUTPUT
    VO_Value : REAL;
    VO_Error : BOOL;
  END_VAR
  VAR
    L_Last_Good_Value : REAL;
    L_First_Valid : BOOL := FALSE;
  END_VAR

            IF VI_Value >= VI_Min_Valid AND VI_Value <= VI_Max_Valid THEN
    VO_Error := FALSE;
    VO_Value := VI_Value;
    L_Last_Good_Value := VI_Value;
    L_First_Valid := TRUE;
ELSE
    VO_Error := TRUE;
    IF VI_Fallback_Mode = 1 OR NOT L_First_Valid THEN
        VO_Value := VI_Default_Value;
    ELSE
        VO_Value := L_Last_Good_Value;
    END_IF;
END_IF;
// >>> BULK_SYNC_ANCHOR: FB_Analog_Validator <<<
          
END_FUNCTION_BLOCK

FUNCTION_BLOCK FB_Distributed_Runtime_Continuity
  VAR_INPUT
    VI_Enable : BOOL;
    VI_System_Time_MS : UDINT;
  END_VAR
  VAR
    L_i : INT;
    L_Node : ST_Distributed_Runtime_Node_State;
    L_Any_Offline : BOOL;
    L_Any_Degraded : BOOL;
    L_Split_Brain : BOOL;
    L_Finalized_Runtime_Continuity : BOOL;
  END_VAR

            IF NOT VI_Enable THEN
    GVL_Distributed_Runtime.G_Runtime_Valid := FALSE;
    RETURN;
END_IF;

// Finalized runtime continuity proof chain.
L_Finalized_Runtime_Continuity :=
    GVL_SEMANTIC_PROGRESS.Semantic_Forward_Progress_Valid
    AND GVL_SEMANTIC_PROGRESS.Semantic_Execution_Continuity_OK
    AND NOT GVL_SEMANTIC_PROGRESS.Semantic_Progress_Lease_Expired
    AND NOT GVL_SEMANTIC_PROGRESS.Semantic_Progress_Quarantine_Active
    AND GVL_RUNTIME_SNAPSHOT.Snapshot_Frozen
    AND GVL_RUNTIME_SNAPSHOT.Snapshot_Publication_Allowed
    AND GVL_RUNTIME_SNAPSHOT.Snapshot_Copy_Valid
    AND GVL_RUNTIME_SNAPSHOT.Snapshot_Isolation_Valid
    AND NOT GVL_RUNTIME_SNAPSHOT.Snapshot_Mutation_Detected
    AND GVL_DISTRIBUTED_SNAPSHOT.Distributed_Publication_Reconciled
    AND GVL_DISTRIBUTED_SNAPSHOT.Distributed_Publication_Freeze_Valid
    AND GVL_DISTRIBUTED_SNAPSHOT.Distributed_Snapshot_Consistent
    AND GVL_DISTRIBUTED_COMMIT.Distributed_Commit_Valid
    AND GVL_DISTRIBUTED_COMMIT.Publication_Prepare_Valid
    AND GVL_DISTRIBUTED_COMMIT.Publication_Commit_Confirmed
    AND NOT GVL_DISTRIBUTED_COMMIT.Peer_Commit_Mismatch
    AND NOT GVL_DISTRIBUTED_COMMIT.Commit_Lease_Expired
    AND GVL_OUTPUT_EPOCH.Output_Publication_Valid
    AND GVL_OUTPUT_EPOCH.Output_Runtime_Epoch_Valid
    AND NOT GVL_OUTPUT_EPOCH.Output_Lease_Expired
    AND NOT GVL_OUTPUT_EPOCH.Output_Forced_Safe_Decay
    AND GVL_COMMAND_VERIFY.PreOutput_Barrier_OK
    AND NOT GVL_COMMAND_VERIFY.PreOutput_Block_IO;

// Local node authoritative runtime state.
GVL_Distributed_Runtime.G_Local_Node_State.Runtime_Valid := TRUE;
GVL_Distributed_Runtime.G_Local_Node_State.Runtime_System_Time_MS :=
    VI_System_Time_MS;

GVL_Distributed_Runtime.G_Local_Node_State.Node_Online :=
    L_Finalized_Runtime_Continuity;

GVL_Distributed_Runtime.G_Local_Node_State.Restart_Continuity_Valid :=
    GVL_Runtime_Restart_Continuity.G_Runtime_Valid
    AND L_Finalized_Runtime_Continuity;

GVL_Distributed_Runtime.G_Local_Node_State.Quarantine_State_Replicated :=
    NOT GVL_Config_Activation.G_Config_Quarantine_Active
    AND L_Finalized_Runtime_Continuity;

GVL_Distributed_Runtime.G_Local_Node_State.Recovery_State_Replicated :=
    GVL_Water_Recovery_Runtime.G_Runtime_Valid
    AND L_Finalized_Runtime_Continuity;

GVL_Distributed_Runtime.G_Local_Node_State.Authority_Allowed :=
    NOT GVL_COMMAND_VERIFY.PreOutput_Block_IO
    AND L_Finalized_Runtime_Continuity;

GVL_Distributed_Runtime.G_Local_Node_State.Replication_Healthy :=
    L_Finalized_Runtime_Continuity;

FOR L_i := 1 TO 8 DO

    L_Node := GVL_Distributed_Runtime.G_Remote_Node_State[L_i];

    IF L_Node.Runtime_Valid THEN

        IF NOT L_Node.Node_Online THEN
            L_Any_Offline := TRUE;
        END_IF;

        IF L_Node.Node_Degraded
           OR L_Node.Node_Quarantined THEN

            L_Any_Degraded := TRUE;

        END_IF;

        IF L_Node.Authority_Master
           AND GVL_Distributed_Runtime.G_Local_Node_State.Authority_Master THEN

            L_Split_Brain := TRUE;

        END_IF;

    END_IF;

END_FOR;

IF NOT L_Finalized_Runtime_Continuity THEN
    L_Any_Degraded := TRUE;
END_IF;

GVL_Distributed_Runtime.G_Any_Remote_Node_Offline :=
    L_Any_Offline;

GVL_Distributed_Runtime.G_Any_Remote_Node_Degraded :=
    L_Any_Degraded;

GVL_Distributed_Runtime.G_Split_Brain_Suspected :=
    L_Split_Brain;

GVL_Distributed_Runtime.G_Distributed_Replication_Healthy :=
    NOT L_Any_Offline
    AND L_Finalized_Runtime_Continuity;

GVL_Distributed_Runtime.G_Distributed_Authority_Healthy :=
    NOT L_Split_Brain
    AND L_Finalized_Runtime_Continuity;

GVL_Distributed_Runtime.G_Runtime_Valid := TRUE;
GVL_Distributed_Runtime.G_Last_Update_MS := VI_System_Time_MS;

IF NOT L_Finalized_Runtime_Continuity THEN
    GVL_Distributed_Runtime.G_Status_Code := 4;
    GVL_Distributed_Runtime.G_Status_Text :=
        'Distributed finalized continuity invalid';
ELSIF L_Split_Brain THEN
    GVL_Distributed_Runtime.G_Status_Code := 3;
    GVL_Distributed_Runtime.G_Status_Text :=
        'Distributed split-brain suspected';
ELSIF L_Any_Degraded THEN
    GVL_Distributed_Runtime.G_Status_Code := 2;
    GVL_Distributed_Runtime.G_Status_Text :=
        'Distributed degraded node detected';
ELSIF L_Any_Offline THEN
    GVL_Distributed_Runtime.G_Status_Code := 1;
    GVL_Distributed_Runtime.G_Status_Text :=
        'Distributed offline node detected';
ELSE
    GVL_Distributed_Runtime.G_Status_Code := 0;
    GVL_Distributed_Runtime.G_Status_Text :=
        'Distributed runtime continuity healthy';
END_IF;
          
END_FUNCTION_BLOCK

FUNCTION_BLOCK FB_Heating_Demand_Map
  VAR_INPUT
    VI_Zone_Valves : ARRAY[1..GVL_CONSTANTS.C_MAX_HEATING_CIRCUITS] OF BOOL;
    VI_Zone_Configs : ARRAY[1..GVL_CONSTANTS.C_MAX_HEATING_CIRCUITS] OF ST_FloorHeating_Circuit_Config;
  END_VAR
  VAR_OUTPUT
    VO_Manifold_Demand_Map : ARRAY[1..GVL_CONSTANTS.C_MAX_MANIFOLDS] OF BOOL;
  END_VAR
  VAR
    L_i : INT;
    L_Manifold_ID : INT;
  END_VAR

            FOR L_i := 1 TO GVL_CONSTANTS.C_MAX_MANIFOLDS DO
    VO_Manifold_Demand_Map[L_i] := FALSE;
END_FOR;

FOR L_i := 1 TO GVL_CONSTANTS.C_MAX_HEATING_CIRCUITS DO
    IF VI_Zone_Valves[L_i] THEN
        L_Manifold_ID := VI_Zone_Configs[L_i].manifold_id;
        IF L_Manifold_ID >= 1 AND L_Manifold_ID <= GVL_CONSTANTS.C_MAX_MANIFOLDS THEN
            VO_Manifold_Demand_Map[L_Manifold_ID] := TRUE;
        END_IF;
    END_IF;
END_FOR;

// >>> BULK_SYNC_ANCHOR: FB_Heating_Demand_Map <<<
          
END_FUNCTION_BLOCK

FUNCTION_BLOCK FB_Access_Output_Projection
  VAR_INPUT
    VI_Lock_1_Open : BOOL;
    VI_Lock_1_Close : BOOL;
    VI_Lock_2_Open : BOOL;
    VI_Lock_2_Close : BOOL;
    VI_Gate_Open : BOOL;
    VI_Wicket_Open : BOOL;
  END_VAR

            GVL_ACCESS_OUTPUT.DO_Lock_1_Open := VI_Lock_1_Open;
GVL_ACCESS_OUTPUT.DO_Lock_1_Close := VI_Lock_1_Close;
GVL_ACCESS_OUTPUT.DO_Lock_2_Open := VI_Lock_2_Open;
GVL_ACCESS_OUTPUT.DO_Lock_2_Close := VI_Lock_2_Close;
GVL_ACCESS_OUTPUT.DO_Gate_Open := VI_Gate_Open;
GVL_ACCESS_OUTPUT.DO_Wicket_Open := VI_Wicket_Open;

// >>> BULK_SYNC_ANCHOR: FB_Access_Output_Projection <<<
          
END_FUNCTION_BLOCK

FUNCTION_BLOCK FB_PLC_Heartbeat
  VAR_INPUT
    VI_Local_ID : BYTE;
    VI_System_Time : UDINT;
    VI_Remote_Pulse : BOOL;
    VI_Remote_Is_Active : BOOL;
    VI_Gateway_Ping_OK : BOOL;
  END_VAR
  VAR_OUTPUT
    VO_Is_Active : BOOL;
    VO_RTT_MS : UDINT;
    VO_Loss_Count : UDINT;
    VO_Max_RTT : UDINT;
  END_VAR
  VAR
    L_Last_Pulse : BOOL;
    L_Last_Pulse_Time : UDINT;
    L_Timeout : UDINT := 500;
    L_Pulse_Send_Time : UDINT;
    L_Last_Loss_Time : UDINT;
    L_Elapsed_Time : UDINT;
  END_VAR

            // Вспомогательная функция для безопасного вычисления разницы времени
L_Elapsed_Time := (VI_System_Time - L_Last_Pulse_Time);

// 1. Мониторинг "сердцебиения" и расчет сетевых задержек (ТЗ 8.4)
IF VI_Remote_Pulse <> L_Last_Pulse THEN
    // Вычисляем время между изменениями сигнала
    VO_RTT_MS := L_Elapsed_Time;
    // Фиксируем пиковые задержки для диагностики сети
    IF VO_RTT_MS > VO_Max_RTT THEN VO_Max_RTT := VO_RTT_MS; END_IF;
    L_Last_Pulse := VI_Remote_Pulse;
    L_Last_Pulse_Time := VI_System_Time;
    L_Elapsed_Time := 0; // Сбрасываем после обновления
END_IF;

// Подсчет статистики потерь связи (ТЗ 8.4)
IF L_Elapsed_Time > L_Timeout THEN
    IF (VI_System_Time - L_Last_Loss_Time) >= 1000 THEN
        VO_Loss_Count := VO_Loss_Count + 1;
        L_Last_Loss_Time := VI_System_Time;
    END_IF;
ELSE
    L_Last_Loss_Time := VI_System_Time;
END_IF;

// 2. Логика определения роли (Active/Standby) и предотвращение Split-Brain (ТЗ 8.3)
// Уровень 1: Проверка наличия связи с партнером
IF L_Elapsed_Time < L_Timeout THEN
    // Связь есть: Договариваемся о ролях на основе приоритета ID
    IF VI_Local_ID = 1 THEN
        VO_Is_Active := TRUE; // ПЛК А всегда активен при наличии связи
    ELSE
        VO_Is_Active := NOT VI_Remote_Is_Active; // ПЛК B активен только если А не активен
    END_IF;
ELSE
    // Связи нет: Пытаемся определить, кто из нас "живее"
    // Уровень 3: Если связи с партнером нет, проверяем доступность внешнего шлюза
    IF VI_Local_ID = 1 THEN
        // ПЛК А становится активным всегда при потере связи с партнером (fallback)
        VO_Is_Active := TRUE;
    ELSE
        // ПЛК B ждет таймаут удержания роли (2 секунды), прежде чем стать активным
        IF L_Elapsed_Time >= 2000 THEN
            // ПЛК B берет управление если он видит шлюз, а связи с А нет.
            // Если шлюз недоступен, B ждет дольше (fallback).
            IF VI_Gateway_Ping_OK THEN
                VO_Is_Active := TRUE;
            ELSIF L_Elapsed_Time >= 5000 THEN
                VO_Is_Active := TRUE; // Fallback: ПЛК А мертв и шлюз мертв
            ELSE
                VO_Is_Active := FALSE;
            END_IF;
        ELSE
            VO_Is_Active := FALSE;
        END_IF;
    END_IF;
END_IF;
          
END_FUNCTION_BLOCK

FUNCTION_BLOCK FB_Vent_Output_Projection
  VAR_INPUT
    VI_Supply_Fans : ARRAY[1..GVL_CONSTANTS.C_MAX_SUPPLY_FANS] OF BYTE;
    VI_Exhaust_Fans : ARRAY[1..GVL_CONSTANTS.C_MAX_EXHAUST_FANS] OF BYTE;
  END_VAR
  VAR
    L_i : INT;
  END_VAR

            // Convert ventilation manager BYTE outputs directly into IO-ready projection.
// PRG_Ventilation no longer needs to publish fan actuator values through GVL_STATE.

FOR L_i := 1 TO GVL_CONSTANTS.C_MAX_SUPPLY_FANS DO
    GVL_VENT_OUTPUT.AO_Supply_Fans[L_i] := BYTE_TO_UINT(VI_Supply_Fans[L_i]) * 10;
END_FOR;

FOR L_i := 1 TO GVL_CONSTANTS.C_MAX_EXHAUST_FANS DO
    GVL_VENT_OUTPUT.AO_Exhaust_Fans[L_i] := BYTE_TO_UINT(VI_Exhaust_Fans[L_i]) * 10;
END_FOR;

// >>> BULK_SYNC_ANCHOR: FB_Vent_Output_Projection <<<
          
END_FUNCTION_BLOCK

FUNCTION_BLOCK FB_System_Health_Orchestrator
  VAR_OUTPUT
    VO_First_Fault_Active : BOOL;
    VO_First_Fault_Type : INT;
    VO_First_Fault_Source : INT;
    VO_System_Severity : E_System_Severity;
    VO_Root_Cause : E_System_Root_Cause;
    VO_Watchdog_Fault : BOOL;
  END_VAR
  VAR
    fbSafety : FB_Safety_Manager;
    fbWatchdog : FB_Watchdog;
    fbSystemHealth : FB_System_Health;
    fbStateManager : FB_State_Manager;
    fbHMIInterface : FB_HMI_Interface;
    fbFaultLogger : FB_Fault_Logger;
  END_VAR

            // ==============================================================================
// System health orchestrator helper
//
// Internal helper for PRG_System.
// Owns safety latch update, watchdog, system health aggregation,
// system mode calculation, HMI/fault publication, diagnostic exports,
// and human-readable mode/cause text projection.
// ==============================================================================



fbSafety(
    VI_Gas_Alarm := GVL_HEALTH_BRIDGE.G_Gas_Detected OR GVL_HEALTH_BRIDGE.G_CO_Alarm_Level,
    VI_Leak_Alarm := GVL_HEALTH_BRIDGE.G_Leak_Detected,
    VI_Smoke_Alarm := GVL_HEALTH_BRIDGE.G_Smoke_Detected,
    VI_Reset := GVL_COMMAND.G_Reset_Errors,
    VO_Gas_Latched => GVL_STATE.G_Safety_Gas_Latched,
    VO_Leak_Latched => GVL_STATE.G_Safety_Leak_Latched,
    VO_Smoke_Latched => GVL_STATE.G_Safety_Smoke_Latched,
    VO_Emergency_Stop => GVL_STATE.G_Safety_Emergency_Stop
);

GVL_STATE.G_Freeze_Hardware_Degraded := GVL_STATUS.G_Diagnostics.Backup_Pump_Fault OR GVL_STATUS.G_Diagnostics.Electric_Heater_Fault;
GVL_STATE.G_Freeze_Hardware_Failed := GVL_STATUS.G_Diagnostics.Backup_Pump_Fault AND GVL_STATUS.G_Diagnostics.Electric_Heater_Fault;

fbWatchdog(
    VI_System_Time_MS := GVL_STATUS.G_System_Time_MS
);

fbSystemHealth(
    VI_Smoke_Detected := GVL_HEALTH_BRIDGE.G_Smoke_Detected OR GVL_STATE.G_Safety_Smoke_Latched,
    VI_Gas_Detected := GVL_HEALTH_BRIDGE.G_Gas_Detected OR GVL_STATE.G_Safety_Gas_Latched,
    VI_CO_Warning_Level := GVL_HEALTH_BRIDGE.G_CO_Warning_Level,
    VI_CO_Alarm_Level := GVL_HEALTH_BRIDGE.G_CO_Alarm_Level,
    VI_Leak_Detected := GVL_HEALTH_BRIDGE.G_Leak_Detected OR GVL_STATE.G_Safety_Leak_Latched,
    VI_Sensor_Fault := GVL_STATE.G_Heating_Sensor_Fault OR GVL_STATE.G_DHW_Sensor_Fault OR GVL_STATUS.G_Diagnostics.Manifold_Pressure_Fault_Active OR GVL_STATUS.G_Diagnostics.Manifold_Current_Fault_Active OR GVL_STATUS.G_Diagnostics.Manifold_Return_Temp_Fault_Active,
    VI_IO_Offline := GVL_STATE.G_Heating_IO_Fault OR GVL_STATE.G_DHW_IO_Fault OR GVL_STATE.G_Ventilation_IO_Fault OR GVL_STATE.G_Lighting_IO_Fault,
    VI_Comm_Fault := GVL_STATE.G_Access_Comm_Fault,
    VI_Watchdog_Fault := fbWatchdog.VO_Watchdog_Fault,
    VI_Subsystem_Fault := GVL_STATE.G_Heating_Subsystem_Degraded OR GVL_STATE.G_DHW_Subsystem_Degraded OR GVL_STATE.G_Ventilation_Subsystem_Degraded OR GVL_STATUS.G_Diagnostics.Manifold_Pressure_Fault_Active OR GVL_STATUS.G_Diagnostics.Manifold_Current_Fault_Active OR GVL_STATUS.G_Diagnostics.Manifold_Return_Temp_Fault_Active
);

fbStateManager(
    VI_System_Severity := fbSystemHealth.VO_System_Severity,
    VI_Root_Cause := fbSystemHealth.VO_Root_Cause,
    VI_Freeze_Risk := GVL_STATE.G_Safety_Freeze_Risk
);

fbHMIInterface(
    VI_Severity := fbSystemHealth.VO_System_Severity,
    VI_RootCause := fbSystemHealth.VO_Root_Cause,
    VI_Status_Msg := fbStateManager.VO_Status_Msg
);

fbFaultLogger(
    VI_Severity := fbSystemHealth.VO_System_Severity,
    VI_RootCause := fbSystemHealth.VO_Root_Cause,
    VI_Time_MS := GVL_STATUS.G_System_Time_MS
);

GVL_STATUS.G_System_Mode_Msg := fbStateManager.VO_Status_Msg;

GVL_STATUS.G_Diagnostics.Sensor_Fault :=
    GVL_STATE.G_Heating_Sensor_Fault OR
    GVL_STATE.G_DHW_Sensor_Fault OR
    GVL_STATUS.G_Diagnostics.Manifold_Pressure_Fault_Active OR
    GVL_STATUS.G_Diagnostics.Manifold_Current_Fault_Active OR
    GVL_STATUS.G_Diagnostics.Manifold_Return_Temp_Fault_Active;

GVL_STATUS.G_Diagnostics.IO_Offline :=
    GVL_STATE.G_Heating_IO_Fault OR
    GVL_STATE.G_DHW_IO_Fault OR
    GVL_STATE.G_Ventilation_IO_Fault OR
    GVL_STATE.G_Lighting_IO_Fault;

GVL_STATUS.G_Diagnostics.Subsystem_Degraded :=
    GVL_STATE.G_Heating_Subsystem_Degraded OR
    GVL_STATE.G_DHW_Subsystem_Degraded OR
    GVL_STATE.G_Ventilation_Subsystem_Degraded OR
    GVL_STATUS.G_Diagnostics.Manifold_Pressure_Fault_Active OR
    GVL_STATUS.G_Diagnostics.Manifold_Current_Fault_Active OR
    GVL_STATUS.G_Diagnostics.Manifold_Return_Temp_Fault_Active;

GVL_GATEWAY.G_Gateway_HMI_Status_Message := fbHMIInterface.VO_HMI_Status_Text;
IF fbFaultLogger.VO_Last_Event_Text <> '' THEN
    GVL_HEALTH_BRIDGE.G_Last_Fault_Event_Text := fbFaultLogger.VO_Last_Event_Text;
END_IF;

GVL_STATE.G_System_Mode := fbStateManager.VO_System_Mode;

CASE GVL_STATE.G_System_Mode OF
    E_System_Operating_Mode.MODE_SAFE_STOP:
        GVL_STATE.G_System_Mode_Text := 'SAFE_STOP';

    E_System_Operating_Mode.MODE_FREEZE_PROTECTION:
        GVL_STATE.G_System_Mode_Text := 'FREEZE_PROTECTION';

    E_System_Operating_Mode.MODE_DEGRADED:
        GVL_STATE.G_System_Mode_Text := 'DEGRADED';

    ELSE
        GVL_STATE.G_System_Mode_Text := 'NORMAL';
END_CASE;

CASE fbSystemHealth.VO_Root_Cause OF
    E_System_Root_Cause.ROOT_FIRE:
        GVL_STATUS.G_System_Mode_Cause := 'Пожар/дым';
    E_System_Root_Cause.ROOT_GAS_LEAK:
        GVL_STATUS.G_System_Mode_Cause := 'Утечка газа';
    E_System_Root_Cause.ROOT_CO_CRITICAL:
        GVL_STATUS.G_System_Mode_Cause := 'Критический CO';
    E_System_Root_Cause.ROOT_CO_WARNING:
        GVL_STATUS.G_System_Mode_Cause := 'Повышенный CO';
    E_System_Root_Cause.ROOT_WATER_LEAK:
        GVL_STATUS.G_System_Mode_Cause := 'Протечка воды';
    E_System_Root_Cause.ROOT_WATCHDOG_FAULT:
        GVL_STATUS.G_System_Mode_Cause := 'Ошибка watchdog';
    E_System_Root_Cause.ROOT_IO_OFFLINE:
        GVL_STATUS.G_System_Mode_Cause := 'Недоступен модуль IO';
    E_System_Root_Cause.ROOT_COMM_FAULT:
        GVL_STATUS.G_System_Mode_Cause := 'Ошибка связи';
    E_System_Root_Cause.ROOT_SENSOR_FAULT:
        GVL_STATUS.G_System_Mode_Cause := 'Ошибка датчика';
    E_System_Root_Cause.ROOT_SUBSYSTEM_FAULT:
        GVL_STATUS.G_System_Mode_Cause := 'Ошибка подсистемы';
    ELSE
        GVL_STATUS.G_System_Mode_Cause := 'Аварийные режимы отсутствуют';
END_CASE;

VO_First_Fault_Active := fbSystemHealth.VO_First_Fault_Active;
VO_First_Fault_Type := fbSystemHealth.VO_First_Fault_Type;
VO_First_Fault_Source := fbSystemHealth.VO_First_Fault_Source;
VO_System_Severity := fbSystemHealth.VO_System_Severity;
VO_Root_Cause := fbSystemHealth.VO_Root_Cause;
VO_Watchdog_Fault := fbWatchdog.VO_Watchdog_Fault;

GVL_STATUS.G_System_Mode_Msg := fbStateManager.VO_Status_Msg;

// >>> BULK_SYNC_ANCHOR: FB_System_Health_Orchestrator <<<
          
END_FUNCTION_BLOCK

FUNCTION_BLOCK FB_Scenario_Transition_Controller
  VAR_INPUT
    VI_System_Time : UDINT;
    VI_Start_Time : UDINT;
    VI_Duration : UDINT;
    VI_Start_Value : REAL;
    VI_End_Value : REAL;
  END_VAR
  VAR_OUTPUT
    VO_Current_Value : REAL;
    VO_Transition_Done : BOOL;
  END_VAR
  VAR
    L_Elapsed : UDINT;
    L_Progress : REAL;
  END_VAR

            L_Elapsed := (SEL(VI_System_Time >= VI_Start_Time, VI_System_Time - VI_Start_Time, (4294967295 - VI_Start_Time) + VI_System_Time + 1));

IF L_Elapsed >= VI_Duration OR VI_Duration = 0 THEN
    VO_Current_Value := VI_End_Value;
    VO_Transition_Done := TRUE;
ELSE
    L_Progress := UDINT_TO_REAL(L_Elapsed) / UDINT_TO_REAL(VI_Duration);
    VO_Current_Value := VI_Start_Value + (VI_End_Value - VI_Start_Value) * L_Progress;
    VO_Transition_Done := FALSE;
END_IF;
          
END_FUNCTION_BLOCK

FUNCTION_BLOCK FB_Heating_Adaptive_Target
  VAR_INPUT
    VI_Base_Target_Supply_Temp : REAL;
    VI_Global_Target_Temperature : REAL;
  END_VAR
  VAR_OUTPUT
    VO_Target_Supply_Temp : REAL;
    VO_Adaptive_Correction : REAL;
    VO_Adaptive_Effective_Delta : REAL;
    VO_Adaptive_Max_Delta : REAL;
  END_VAR
  VAR_IN_OUT
    VI_Zone_Configs : ARRAY[1..GVL_CONSTANTS.C_MAX_HEATING_CIRCUITS] OF ST_FloorHeating_Circuit_Config;
    VI_Floor_Temps : ARRAY[1..GVL_CONSTANTS.C_MAX_HEATING_CIRCUITS] OF REAL;
    VI_Room_Temps : ARRAY[1..GVL_CONSTANTS.C_MAX_ZONES] OF REAL;
  END_VAR
  VAR
    L_Adaptive_Zone_i : INT;
    L_Zone_Index : INT;
    L_Adaptive_Delta : REAL;
    L_Adaptive_Weighted_Sum : REAL;
    L_Adaptive_Weight_Total : REAL;
    L_Adaptive_Weight : REAL;
  END_VAR

            // ==============================================================================
// Adaptive target calculation for heating supply temperature
// ==============================================================================



VO_Target_Supply_Temp := VI_Base_Target_Supply_Temp;
VO_Adaptive_Max_Delta := 0.0;
L_Adaptive_Weighted_Sum := 0.0;
L_Adaptive_Weight_Total := 0.0;
VO_Adaptive_Effective_Delta := 0.0;
VO_Adaptive_Correction := 0.0;

IF VI_Global_Target_Temperature > 0.0 THEN
    VO_Target_Supply_Temp := VI_Global_Target_Temperature;
END_IF;

FOR L_Adaptive_Zone_i := 1 TO GVL_CONSTANTS.C_MAX_HEATING_CIRCUITS DO
    L_Zone_Index := VI_Zone_Configs[L_Adaptive_Zone_i].zone;

    IF (L_Zone_Index >= 1) AND (L_Zone_Index <= GVL_CONSTANTS.C_MAX_ZONES) THEN
        CASE VI_Zone_Configs[L_Adaptive_Zone_i].control_type OF
            0:
                L_Adaptive_Delta :=
                    VI_Zone_Configs[L_Adaptive_Zone_i].design_temp -
                    VI_Floor_Temps[L_Adaptive_Zone_i];
                L_Adaptive_Weight := 0.6;
            1, 2:
                L_Adaptive_Delta :=
                    VI_Zone_Configs[L_Adaptive_Zone_i].design_temp -
                    VI_Room_Temps[L_Zone_Index];
                L_Adaptive_Weight := 1.0;
            ELSE
                L_Adaptive_Delta :=
                    VI_Zone_Configs[L_Adaptive_Zone_i].design_temp -
                    VI_Room_Temps[L_Zone_Index];
                L_Adaptive_Weight := 0.8;
        END_CASE;

        IF L_Zone_Index <= 4 THEN
            L_Adaptive_Weight := L_Adaptive_Weight * 1.2;
        ELSIF L_Zone_Index >= 9 THEN
            L_Adaptive_Weight := L_Adaptive_Weight * 0.7;
        END_IF;

        IF L_Adaptive_Weight > 2.0 THEN
            L_Adaptive_Weight := 2.0;
        ELSIF L_Adaptive_Weight < 0.2 THEN
            L_Adaptive_Weight := 0.2;
        END_IF;

        IF L_Adaptive_Delta > VO_Adaptive_Max_Delta THEN
            VO_Adaptive_Max_Delta := L_Adaptive_Delta;
        END_IF;

        L_Adaptive_Weighted_Sum := L_Adaptive_Weighted_Sum + (L_Adaptive_Delta * L_Adaptive_Weight);
        L_Adaptive_Weight_Total := L_Adaptive_Weight_Total + L_Adaptive_Weight;
    END_IF;
END_FOR;

IF L_Adaptive_Weight_Total > 0.0 THEN
    VO_Adaptive_Effective_Delta := L_Adaptive_Weighted_Sum / L_Adaptive_Weight_Total;
END_IF;

IF VO_Adaptive_Effective_Delta > 1.5 THEN
    VO_Adaptive_Correction := 2.0;
ELSIF VO_Adaptive_Effective_Delta > 0.7 THEN
    VO_Adaptive_Correction := 1.0;
ELSIF VO_Adaptive_Effective_Delta < -1.5 THEN
    VO_Adaptive_Correction := -2.0;
ELSIF VO_Adaptive_Effective_Delta < -0.7 THEN
    VO_Adaptive_Correction := -1.0;
ELSE
    VO_Adaptive_Correction := 0.0;
END_IF;

IF VO_Adaptive_Max_Delta > 2.5 AND VO_Adaptive_Correction < 2.0 THEN
    VO_Adaptive_Correction := 2.0;
END_IF;

VO_Target_Supply_Temp := VO_Target_Supply_Temp + VO_Adaptive_Correction;

IF VO_Target_Supply_Temp < 20.0 THEN
    VO_Target_Supply_Temp := 20.0;
ELSIF VO_Target_Supply_Temp > 45.0 THEN
    VO_Target_Supply_Temp := 45.0;
END_IF;

// >>> BULK_SYNC_ANCHOR: FB_Heating_Adaptive_Target <<<
          
END_FUNCTION_BLOCK

FUNCTION_BLOCK FB_Heating_Policy_Observer
  VAR_INPUT
    VI_Zone_Occupied : ARRAY[1..GVL_CONSTANTS.C_MAX_ZONES] OF BOOL;
    VI_Zone_Last_Motion_TS : ARRAY[1..GVL_CONSTANTS.C_MAX_ZONES] OF UDINT;
    VI_System_Time_MS : UDINT;
    VI_Zone_Permanent_Use : ARRAY[1..GVL_CONSTANTS.C_MAX_ZONES] OF BOOL;
    VI_Zone_Guest_Preheat : ARRAY[1..GVL_CONSTANTS.C_MAX_ZONES] OF BOOL;
    VI_Behavior_Mode : E_Behavior_Mode;
  END_VAR
  VAR_OUTPUT
    VO_Zone_Empty_Duration_MS : ARRAY[1..GVL_CONSTANTS.C_MAX_ZONES] OF UDINT;
    VO_Zone_Policy_Class : ARRAY[1..GVL_CONSTANTS.C_MAX_ZONES] OF INT;
    VO_Zone_Target_Adjustment : ARRAY[1..GVL_CONSTANTS.C_MAX_ZONES] OF REAL;
    VO_Zone_Priority_Bias : ARRAY[1..GVL_CONSTANTS.C_MAX_ZONES] OF REAL;
  END_VAR
  VAR
    L_i : INT;
    L_Long_Threshold : UDINT := 86400000;
    L_Away_Mode : BOOL;
  END_VAR

            L_Away_Mode := (VI_Behavior_Mode = BEHAVIOR_AWAY);

FOR L_i := 1 TO GVL_CONSTANTS.C_MAX_ZONES DO

    // compute empty duration
    IF VI_Zone_Occupied[L_i] THEN
        VO_Zone_Empty_Duration_MS[L_i] := 0;
    ELSE
        VO_Zone_Empty_Duration_MS[L_i] := VI_System_Time_MS - VI_Zone_Last_Motion_TS[L_i];
    END_IF;

    // policy classification
    // Guest/preheat has priority even in AWAY mode.
    IF VI_Zone_Guest_Preheat[L_i] THEN
        VO_Zone_Policy_Class[L_i] := 3; // guest

    ELSIF VI_Zone_Occupied[L_i] THEN
        VO_Zone_Policy_Class[L_i] := 0; // comfort

    ELSIF VI_Zone_Permanent_Use[L_i] AND (NOT L_Away_Mode) THEN
        VO_Zone_Policy_Class[L_i] := 4; // permanent mild eco

    ELSIF VO_Zone_Empty_Duration_MS[L_i] >= L_Long_Threshold THEN
        VO_Zone_Policy_Class[L_i] := 2; // deep eco

    ELSE
        VO_Zone_Policy_Class[L_i] := 1; // mild eco
    END_IF;

    // observe-only target adjustment (no effect yet)
    CASE VO_Zone_Policy_Class[L_i] OF
        0: // comfort
            VO_Zone_Target_Adjustment[L_i] := 0.0;
            VO_Zone_Priority_Bias[L_i] := 1.0;

        1: // mild eco
            VO_Zone_Target_Adjustment[L_i] := -1.0;
            VO_Zone_Priority_Bias[L_i] := 0.8;

        2: // deep eco
            VO_Zone_Target_Adjustment[L_i] := -3.0;
            VO_Zone_Priority_Bias[L_i] := 0.5;

        3: // guest preheat
            VO_Zone_Target_Adjustment[L_i] := 0.0;
            VO_Zone_Priority_Bias[L_i] := 1.5;

        4: // permanent-use mild eco
            VO_Zone_Target_Adjustment[L_i] := -0.5;
            VO_Zone_Priority_Bias[L_i] := 0.9;

    END_CASE;

END_FOR;
          
END_FUNCTION_BLOCK

FUNCTION_BLOCK FB_Safety_Workflow_Manager
  VAR_INPUT
    VI_System_Time_MS : UDINT;
    VI_Water_Selective_Recover : BOOL;
    VI_Gas_Selective_Recover : BOOL;
    VI_Water_Valve_Test_Open : BOOL;
    VI_Water_Valve_Test_Close : BOOL;
    VI_Water_Valve_Test_Confirm : BOOL;
    VI_Gas_Valve_Test_Open : BOOL;
    VI_Gas_Valve_Test_Close : BOOL;
    VI_Gas_Valve_Test_Confirm : BOOL;
  END_VAR
  VAR_OUTPUT
    VO_Water_Selective_Recover_Edge : BOOL;
    VO_Gas_Selective_Recover_Edge : BOOL;
    VO_Water_Valve_Test_Open_Edge : BOOL;
    VO_Water_Valve_Test_Close_Edge : BOOL;
    VO_Water_Valve_Test_Confirm_Edge : BOOL;
    VO_Gas_Valve_Test_Open_Edge : BOOL;
    VO_Gas_Valve_Test_Close_Edge : BOOL;
    VO_Gas_Valve_Test_Confirm_Edge : BOOL;
    VO_Water_Test_Active : BOOL;
    VO_Gas_Test_Active : BOOL;
    VO_Water_Test_Timeout_Close_Required : BOOL;
    VO_Gas_Test_Timeout_Close_Required : BOOL;
  END_VAR
  VAR
    L_CMD_Water_Selective_Recover_Prev : BOOL;
    L_CMD_Gas_Selective_Recover_Prev : BOOL;
    L_CMD_Water_Valve_Test_Open_Prev : BOOL;
    L_CMD_Water_Valve_Test_Close_Prev : BOOL;
    L_CMD_Water_Valve_Test_Confirm_Prev : BOOL;
    L_CMD_Gas_Valve_Test_Open_Prev : BOOL;
    L_CMD_Gas_Valve_Test_Close_Prev : BOOL;
    L_CMD_Gas_Valve_Test_Confirm_Prev : BOOL;
    L_Water_Test_Active : BOOL;
    L_Water_Test_Deadline : UDINT;
    L_Gas_Test_Active : BOOL;
    L_Gas_Test_Deadline : UDINT;
  END_VAR

            VO_Water_Test_Timeout_Close_Required := FALSE;
VO_Gas_Test_Timeout_Close_Required := FALSE;

VO_Water_Selective_Recover_Edge := VI_Water_Selective_Recover AND NOT L_CMD_Water_Selective_Recover_Prev;
VO_Gas_Selective_Recover_Edge := VI_Gas_Selective_Recover AND NOT L_CMD_Gas_Selective_Recover_Prev;
VO_Water_Valve_Test_Open_Edge := VI_Water_Valve_Test_Open AND NOT L_CMD_Water_Valve_Test_Open_Prev;
VO_Water_Valve_Test_Close_Edge := VI_Water_Valve_Test_Close AND NOT L_CMD_Water_Valve_Test_Close_Prev;
VO_Water_Valve_Test_Confirm_Edge := VI_Water_Valve_Test_Confirm AND NOT L_CMD_Water_Valve_Test_Confirm_Prev;
VO_Gas_Valve_Test_Open_Edge := VI_Gas_Valve_Test_Open AND NOT L_CMD_Gas_Valve_Test_Open_Prev;
VO_Gas_Valve_Test_Close_Edge := VI_Gas_Valve_Test_Close AND NOT L_CMD_Gas_Valve_Test_Close_Prev;
VO_Gas_Valve_Test_Confirm_Edge := VI_Gas_Valve_Test_Confirm AND NOT L_CMD_Gas_Valve_Test_Confirm_Prev;

L_CMD_Water_Selective_Recover_Prev := VI_Water_Selective_Recover;
L_CMD_Gas_Selective_Recover_Prev := VI_Gas_Selective_Recover;
L_CMD_Water_Valve_Test_Open_Prev := VI_Water_Valve_Test_Open;
L_CMD_Water_Valve_Test_Close_Prev := VI_Water_Valve_Test_Close;
L_CMD_Water_Valve_Test_Confirm_Prev := VI_Water_Valve_Test_Confirm;
L_CMD_Gas_Valve_Test_Open_Prev := VI_Gas_Valve_Test_Open;
L_CMD_Gas_Valve_Test_Close_Prev := VI_Gas_Valve_Test_Close;
L_CMD_Gas_Valve_Test_Confirm_Prev := VI_Gas_Valve_Test_Confirm;

IF VO_Water_Valve_Test_Open_Edge THEN
    L_Water_Test_Active := TRUE;
    L_Water_Test_Deadline := VI_System_Time_MS + 60000;
END_IF;

IF L_Water_Test_Active THEN
    IF VI_System_Time_MS >= L_Water_Test_Deadline THEN
        L_Water_Test_Active := FALSE;
        VO_Water_Test_Timeout_Close_Required := TRUE;
    END_IF;
END_IF;

IF VO_Gas_Valve_Test_Open_Edge THEN
    L_Gas_Test_Active := TRUE;
    L_Gas_Test_Deadline := VI_System_Time_MS + 60000;
END_IF;

IF L_Gas_Test_Active THEN
    IF VI_System_Time_MS >= L_Gas_Test_Deadline THEN
        L_Gas_Test_Active := FALSE;
        VO_Gas_Test_Timeout_Close_Required := TRUE;
    END_IF;
END_IF;

VO_Water_Test_Active := L_Water_Test_Active;
VO_Gas_Test_Active := L_Gas_Test_Active;
          
END_FUNCTION_BLOCK

FUNCTION_BLOCK FB_Runtime_Restart_Continuity
  VAR_INPUT
    VI_Enable : BOOL;
    VI_System_Time_MS : UDINT;
    VI_Warm_Restart : BOOL;
  END_VAR
  VAR
    L_State : ST_Runtime_Restart_Continuity_State;
  END_VAR

            IF NOT VI_Enable THEN
    GVL_Runtime_Restart_Continuity.G_Runtime_Valid := FALSE;
    RETURN;
END_IF;

L_State.Runtime_Valid := TRUE;
L_State.Runtime_System_Time_MS := VI_System_Time_MS;

L_State.Warm_Restart_Detected := VI_Warm_Restart;
L_State.Cold_Start_Detected := NOT VI_Warm_Restart;

L_State.Active_Config_Version :=
    GVL_Water_Topology_Config.G_Active_Config_Version;

L_State.Restored_Config_Version :=
    GVL_Runtime_Restart_Continuity.G_Last_Stable_Config_Version;

L_State.Last_Stable_Config_Version :=
    GVL_Runtime_Restart_Continuity.G_Last_Stable_Config_Version;

L_State.Restore_Requested :=
    GVL_Runtime_Restart_Continuity.G_Restore_Request;

L_State.Post_Restart_Validation_Required :=
    GVL_Runtime_Restart_Continuity.G_Post_Restart_Validation_Request;

L_State.Retained_State_Valid := TRUE;
L_State.Topology_Restore_Valid := TRUE;
L_State.Config_Restore_Valid := TRUE;
L_State.Recovery_Restore_Valid := TRUE;
L_State.Quarantine_Restore_Valid := TRUE;

IF L_State.Restore_Requested THEN

    IF L_State.Retained_State_Valid
       AND L_State.Topology_Restore_Valid
       AND L_State.Config_Restore_Valid THEN

        L_State.Restore_Allowed := TRUE;
        L_State.Restore_Completed := TRUE;

        GVL_Config_Activation.G_Config_Quarantine_Active :=
            GVL_Runtime_Restart_Continuity.G_Last_Known_Quarantine_State;

        L_State.Status_Code := 1;
        L_State.Status_Text := 'Runtime continuity restored';

    ELSE

        L_State.Restore_Blocked := TRUE;
        L_State.Safe_Mode_Required := TRUE;
        L_State.Operator_Ack_Required := TRUE;

        L_State.Status_Code := 2;
        L_State.Status_Text := 'Runtime continuity restore blocked';

    END_IF;

ELSIF L_State.Post_Restart_Validation_Required THEN

    IF GVL_Water_Runtime_Hardening.G_Runtime_Valid
       AND GVL_Water_Output_Reconciliation.G_Runtime_Valid
       AND NOT GVL_Water_Output_Reconciliation.G_Any_Conflict_Detected THEN

        L_State.Post_Restart_Validation_OK := TRUE;

        L_State.Status_Code := 0;
        L_State.Status_Text := 'Post-restart validation healthy';

    ELSE

        L_State.Post_Restart_Validation_Failed := TRUE;
        L_State.Safe_Mode_Required := TRUE;

        L_State.Status_Code := 3;
        L_State.Status_Text := 'Post-restart validation failed';

    END_IF;

ELSE

    L_State.Status_Code := 0;
    L_State.Status_Text := 'Runtime restart continuity healthy';

END_IF;

GVL_Runtime_Restart_Continuity.G_Continuity_State := L_State;

GVL_Runtime_Restart_Continuity.G_Runtime_Valid := TRUE;
GVL_Runtime_Restart_Continuity.G_Last_Update_MS := VI_System_Time_MS;
GVL_Runtime_Restart_Continuity.G_Status_Code := L_State.Status_Code;
GVL_Runtime_Restart_Continuity.G_Status_Text := L_State.Status_Text;
          
END_FUNCTION_BLOCK

FUNCTION_BLOCK FB_Heating_Runtime_Event_Reconstruction_Engine
  VAR_INPUT
    VI_Enable : BOOL;
    VI_Node : ST_Heating_Runtime_Causality_Node;
    VI_Edge : ST_Heating_Runtime_Causality_Edge;
    VI_System_Time_MS : UDINT;
  END_VAR
  VAR_OUTPUT
    VO_Event : ST_Heating_Runtime_Blackbox_Event;
  END_VAR

            // ==============================================================================
// Heating runtime event reconstruction engine
// Read-only runtime forensic reconstruction layer.
// ==============================================================================



// ======================================================
// DETERMINISTIC DEFAULTS
// ======================================================
VO_Event.Event_ID := 0;
VO_Event.Event_Active := FALSE;

VO_Event.Runtime_Phase :=
    E_Heating_Runtime_Phase.HRP_DISABLED;

VO_Event.Event_Start_MS := 0;
VO_Event.Event_End_MS := 0;
VO_Event.Event_Duration_MS := 0;

VO_Event.Runtime_Degraded := FALSE;
VO_Event.Runtime_Fault := FALSE;

VO_Event.Cascade_Degraded := FALSE;
VO_Event.Cascade_Boiler_Loss := FALSE;

VO_Event.OpenTherm_Degraded := FALSE;
VO_Event.OpenTherm_Command_Invalid := FALSE;

VO_Event.Sequencing_Invalid := FALSE;
VO_Event.Ownership_Invalid := FALSE;
VO_Event.Synchronization_Invalid := FALSE;

VO_Event.Root_Cause_Candidate := FALSE;
VO_Event.Critical_Path := FALSE;

VO_Event.Status_Code := 0;
VO_Event.Status_Text := 'Heating runtime reconstruction engine disabled';

IF NOT VI_Enable THEN
    RETURN;
END_IF;

// ======================================================
// EVENT RECONSTRUCTION
// ======================================================
VO_Event.Event_ID := VI_System_Time_MS;
VO_Event.Event_Active := VI_Node.Node_Active;

VO_Event.Runtime_Phase :=
    E_Heating_Runtime_Phase.HRP_COMPLETE;

VO_Event.Event_Start_MS := VI_System_Time_MS;
VO_Event.Event_End_MS := VI_System_Time_MS;
VO_Event.Event_Duration_MS := 0;

VO_Event.Runtime_Degraded :=
    VI_Node.Runtime_Degraded;

VO_Event.Runtime_Fault :=
    VI_Node.Runtime_Fault;

VO_Event.Cascade_Degraded :=
    VI_Node.Cascade_Degraded;

VO_Event.Cascade_Boiler_Loss :=
    VI_Node.Cascade_Boiler_Loss;

VO_Event.OpenTherm_Degraded :=
    VI_Node.OpenTherm_Degraded;

VO_Event.OpenTherm_Command_Invalid :=
    VI_Node.OpenTherm_Command_Invalid;

VO_Event.Sequencing_Invalid :=
    VI_Node.Sequencing_Invalid;

VO_Event.Ownership_Invalid :=
    VI_Node.Ownership_Invalid;

VO_Event.Synchronization_Invalid :=
    VI_Node.Synchronization_Invalid;

VO_Event.Root_Cause_Candidate :=
    VI_Node.Root_Cause_Candidate;

VO_Event.Critical_Path :=
    VI_Edge.Critical_Path;

// ======================================================
// STATUS
// ======================================================
IF VO_Event.Root_Cause_Candidate THEN
    VO_Event.Status_Code := 900;
    VO_Event.Status_Text := 'Heating runtime root-cause reconstructed';
ELSE
    VO_Event.Status_Code := 1;
    VO_Event.Status_Text := 'Heating runtime event reconstructed';
END_IF;

// >>> BULK_SYNC_ANCHOR: FB_Heating_Runtime_Event_Reconstruction_Engine <<<
          
END_FUNCTION_BLOCK

FUNCTION_BLOCK FB_Config_Activation_Runtime
  VAR_INPUT
    VI_Enable : BOOL;
    VI_System_Time_MS : UDINT;
  END_VAR
  VAR
    L_i : INT;
    L_State : ST_Config_Activation_State;
    L_Staged_Valid : BOOL;
  END_VAR

            IF NOT VI_Enable THEN
    GVL_Config_Activation.G_Activation_Runtime_Valid := FALSE;
    RETURN;
END_IF;

L_State.Runtime_Valid := TRUE;
L_State.Runtime_System_Time_MS := VI_System_Time_MS;

L_State.Active_Version :=
    GVL_Water_Topology_Config.G_Active_Config_Version;

L_State.Staged_Version :=
    GVL_Config_Activation.G_Staged_Config_Version;

L_State.Previous_Stable_Version :=
    GVL_Config_Activation.G_Last_Stable_Config_Version;

L_State.Activation_Requested :=
    GVL_Config_Activation.G_Activation_Request;

L_State.Rollback_Requested :=
    GVL_Config_Activation.G_Rollback_Request;

L_State.Rollback_Available :=
    GVL_Config_Activation.G_Last_Stable_Config_Version <> 0;

L_Staged_Valid := TRUE;

FOR L_i := 1 TO GVL_CONSTANTS.C_MAX_FLOOD_SENSORS DO

    IF GVL_Config_Activation.G_Staged_Topology_Config[L_i].Primary_Valve_Group_Id = 0 THEN
        L_Staged_Valid := FALSE;
    END_IF;

END_FOR;

L_State.Staged_Config_Valid := L_Staged_Valid;
L_State.Migration_Compatible := TRUE;

IF L_State.Rollback_Requested
   AND L_State.Rollback_Available THEN

    L_State.Rollback_Active := TRUE;
    L_State.Activation_Blocked := TRUE;

    GVL_Config_Activation.G_Config_Quarantine_Active := FALSE;

    L_State.Status_Code := 3;
    L_State.Status_Text := 'Rollback activation active';

ELSIF L_State.Activation_Requested THEN

    IF NOT L_State.Staged_Config_Valid THEN

        L_State.Activation_Blocked := TRUE;
        L_State.Config_Quarantine_Active := TRUE;

        GVL_Config_Activation.G_Config_Quarantine_Active := TRUE;

        L_State.Status_Code := 2;
        L_State.Status_Text := 'Config activation quarantined';

    ELSE

        L_State.Activation_Allowed := TRUE;

        GVL_Water_Topology_Config_Source.G_Source_Version :=
            L_State.Staged_Version;

        FOR L_i := 1 TO GVL_CONSTANTS.C_MAX_FLOOD_SENSORS DO

            GVL_Water_Topology_Config_Source.G_Source_Record[L_i] :=
                GVL_Config_Activation.G_Staged_Topology_Config[L_i];

        END_FOR;

        GVL_Water_Topology_Config_Source.G_Source_Valid := TRUE;
        GVL_Water_Topology_Config_Source.G_Source_Activated_MS := VI_System_Time_MS;

        GVL_Config_Activation.G_Last_Stable_Config_Version :=
            L_State.Staged_Version;

        GVL_Config_Activation.G_Config_Quarantine_Active := FALSE;

        L_State.Status_Code := 1;
        L_State.Status_Text := 'Config activation completed';

    END_IF;

ELSE

    L_State.Status_Code := 0;
    L_State.Status_Text := 'Config activation runtime healthy';

END_IF;

GVL_Config_Activation.G_Activation_State := L_State;

GVL_Config_Activation.G_Activation_Runtime_Valid := TRUE;
GVL_Config_Activation.G_Last_Update_MS := VI_System_Time_MS;
GVL_Config_Activation.G_Status_Code := L_State.Status_Code;
GVL_Config_Activation.G_Status_Text := L_State.Status_Text;
          
END_FUNCTION_BLOCK

FUNCTION_BLOCK FB_Water_Recovery_Runtime
  VAR_INPUT
    VI_Enable : BOOL;
    VI_System_Time_MS : UDINT;
  END_VAR
  VAR
    L_i : INT;
    L_Feedback : ST_Water_Valve_Feedback_State;
    L_State : ST_Water_Recovery_Runtime_State;
    L_Any_Denied : BOOL;
    L_Any_Unsafe : BOOL;
  END_VAR

            IF NOT VI_Enable THEN
    GVL_Water_Recovery_Runtime.G_Runtime_Valid := FALSE;
    RETURN;
END_IF;

FOR L_i := 1 TO GVL_CONSTANTS.C_MAX_FLOOD_SENSORS DO
    L_Feedback := GVL_Water_Valve_Feedback.G_Valve_Feedback_State[L_i];

    L_State.Runtime_Valid := TRUE;
    L_State.Runtime_System_Time_MS := VI_System_Time_MS;
    L_State.Recovery_Requested := GVL_INTENT_SAFETY.I_Water_Selective_Recovery_Allowed;
    L_State.Valve_Degraded := L_Feedback.Valve_Degraded;
    L_State.Confirmation_Healthy := NOT L_Feedback.Feedback_Conflict;
    L_State.Recovery_Target_Valid := L_Feedback.Valve_Group_Id <> 0;

    IF NOT L_State.Recovery_Target_Valid THEN
        L_State.Recovery_Denied := TRUE;
        L_State.Status_Code := 1;
        L_State.Status_Text := 'Recovery target invalid';
    ELSIF L_State.Valve_Degraded THEN
        L_State.Recovery_Denied := TRUE;
        L_State.Unsafe_Recovery_Detected := TRUE;
        L_State.Status_Code := 2;
        L_State.Status_Text := 'Recovery blocked by valve state';
    ELSIF NOT L_State.Confirmation_Healthy THEN
        L_State.Recovery_Denied := TRUE;
        L_State.Status_Code := 3;
        L_State.Status_Text := 'Recovery blocked by confirmation state';
    ELSE
        L_State.Recovery_Allowed := TRUE;
        L_State.Observation_Window_Active := TRUE;
        L_State.Status_Code := 0;
        L_State.Status_Text := 'Recovery governance healthy';
    END_IF;

    GVL_Water_Recovery_Runtime.G_Recovery_State[L_i] := L_State;
    L_Any_Denied := L_Any_Denied OR L_State.Recovery_Denied;
    L_Any_Unsafe := L_Any_Unsafe OR L_State.Unsafe_Recovery_Detected;
END_FOR;

GVL_Water_Recovery_Runtime.G_Any_Recovery_Denied := L_Any_Denied;
GVL_Water_Recovery_Runtime.G_Any_Unsafe_Recovery := L_Any_Unsafe;
GVL_Water_Recovery_Runtime.G_Runtime_Valid := TRUE;
GVL_Water_Recovery_Runtime.G_Last_Update_MS := VI_System_Time_MS;

IF L_Any_Unsafe THEN
    GVL_Water_Recovery_Runtime.G_Status_Code := 2;
    GVL_Water_Recovery_Runtime.G_Status_Text := 'Recovery risk detected';
ELSIF L_Any_Denied THEN
    GVL_Water_Recovery_Runtime.G_Status_Code := 1;
    GVL_Water_Recovery_Runtime.G_Status_Text := 'Recovery governance denied';
ELSE
    GVL_Water_Recovery_Runtime.G_Status_Code := 0;
    GVL_Water_Recovery_Runtime.G_Status_Text := 'Recovery governance healthy';
END_IF;
          
END_FUNCTION_BLOCK

FUNCTION_BLOCK FB_Predictive_Diagnostics_Runtime
  VAR_INPUT
    VI_Enable : BOOL;
    VI_System_Time_MS : UDINT;
  END_VAR
  VAR
    L_i : INT;
    L_State : ST_Predictive_Diagnostics_State;
    L_Feedback : ST_Water_Valve_Feedback_State;
    L_Recovery : ST_Water_Recovery_Runtime_State;
    L_Any_Degrading : BOOL;
    L_Any_Service : BOOL;
    L_Any_Urgent : BOOL;
  END_VAR

            IF NOT VI_Enable THEN
    GVL_Predictive_Diagnostics.G_Runtime_Valid := FALSE;
    RETURN;
END_IF;

FOR L_i := 1 TO GVL_CONSTANTS.C_MAX_FLOOD_SENSORS DO

    L_State := GVL_Predictive_Diagnostics.G_Diagnostics_State[L_i];

    L_Feedback :=
        GVL_Water_Valve_Feedback.G_Valve_Feedback_State[L_i];

    L_Recovery :=
        GVL_Water_Recovery_Runtime.G_Recovery_State[L_i];

    L_State.Runtime_Valid := TRUE;
    L_State.Runtime_System_Time_MS := VI_System_Time_MS;

    L_State.Device_Id := TO_UINT(L_i);
    L_State.Valve_Group_Id := L_Feedback.Valve_Group_Id;

    IF L_Feedback.Feedback_Timeout THEN
        L_State.Timeout_Count := L_State.Timeout_Count + 1;
    END_IF;

    IF L_Feedback.Feedback_Conflict THEN
        L_State.Conflict_Count := L_State.Conflict_Count + 1;
    END_IF;

    IF L_Recovery.Recovery_Denied THEN
        L_State.Recovery_Denied_Count :=
            L_State.Recovery_Denied_Count + 1;
    END_IF;

    L_State.Failure_Count :=
        L_State.Timeout_Count
        + L_State.Conflict_Count
        + L_State.Recovery_Denied_Count;

    // Predictive accumulation model foundation.
    L_State.Wear_Score :=
        TO_REAL(L_State.Failure_Count) * 0.1;

    L_State.Reliability_Score :=
        100.0 - L_State.Wear_Score;

    IF L_State.Reliability_Score < 0.0 THEN
        L_State.Reliability_Score := 0.0;
    END_IF;

    IF L_State.Failure_Count >= 3 THEN

        L_State.Degradation_Accumulating := TRUE;
        L_State.Service_Recommended := TRUE;

    END_IF;

    IF L_State.Failure_Count >= 10 THEN

        L_State.Service_Urgent := TRUE;
        L_State.Predictive_Quarantine_Recommended := TRUE;

    END_IF;

    IF L_State.Conflict_Count >= 2 THEN
        L_State.Intermittent_Fault_Suspected := TRUE;
    END_IF;

    IF L_State.Service_Urgent THEN

        L_State.Status_Code := 2;
        L_State.Status_Text :=
            'Urgent predictive maintenance required';

    ELSIF L_State.Service_Recommended THEN

        L_State.Status_Code := 1;
        L_State.Status_Text :=
            'Predictive maintenance recommended';

    ELSE

        L_State.Status_Code := 0;
        L_State.Status_Text :=
            'Predictive diagnostics healthy';

    END_IF;

    GVL_Predictive_Diagnostics.G_Diagnostics_State[L_i] :=
        L_State;

    L_Any_Degrading :=
        L_Any_Degrading
        OR L_State.Degradation_Accumulating;

    L_Any_Service :=
        L_Any_Service
        OR L_State.Service_Recommended;

    L_Any_Urgent :=
        L_Any_Urgent
        OR L_State.Service_Urgent;

END_FOR;

GVL_Predictive_Diagnostics.G_Any_Degradation_Accumulating :=
    L_Any_Degrading;

GVL_Predictive_Diagnostics.G_Any_Service_Recommended :=
    L_Any_Service;

GVL_Predictive_Diagnostics.G_Any_Urgent_Service :=
    L_Any_Urgent;

GVL_Predictive_Diagnostics.G_Runtime_Valid := TRUE;
GVL_Predictive_Diagnostics.G_Last_Update_MS := VI_System_Time_MS;

IF L_Any_Urgent THEN
    GVL_Predictive_Diagnostics.G_Status_Code := 2;
    GVL_Predictive_Diagnostics.G_Status_Text :=
        'Urgent predictive maintenance required';
ELSIF L_Any_Service THEN
    GVL_Predictive_Diagnostics.G_Status_Code := 1;
    GVL_Predictive_Diagnostics.G_Status_Text :=
        'Predictive maintenance recommended';
ELSE
    GVL_Predictive_Diagnostics.G_Status_Code := 0;
    GVL_Predictive_Diagnostics.G_Status_Text :=
        'Predictive diagnostics runtime healthy';
END_IF;
          
END_FUNCTION_BLOCK

FUNCTION_BLOCK FB_Command_Deduplication
  VAR_INPUT
    VI_Command_ID : UDINT;
    VI_Command_Type : E_Gateway_Command_Type;
    VI_Command_Value : REAL;
    VI_System_Time_MS : UDINT;
  END_VAR
  VAR_OUTPUT
    VO_Is_New_Command : BOOL;
    VO_Processed_ID : UDINT;
  END_VAR
  VAR
    L_Processed_History : ARRAY[0..GVL_CONSTANTS.C_MAX_DEDUPLICATION_HISTORY-1] OF UDINT;
    L_Processed_Times : ARRAY[0..GVL_CONSTANTS.C_MAX_DEDUPLICATION_HISTORY-1] OF UDINT;
    L_History_Index : INT := 0;
    L_i : INT;
    L_Found : BOOL;
  END_VAR

            // Check if command ID is already in history
L_Found := FALSE;
FOR L_i := 0 TO GVL_CONSTANTS.C_MAX_DEDUPLICATION_HISTORY-1 DO
    IF L_Processed_History[L_i] = VI_Command_ID AND VI_Command_ID <> 0 THEN
        // Check if the command is not too old (e.g., 1 hour = 3600000 ms)
        IF (VI_System_Time_MS - L_Processed_Times[L_i]) < 3600000 THEN
            L_Found := TRUE;
            EXIT;
        END_IF;
    END_IF;
END_FOR;

IF NOT L_Found AND VI_Command_ID <> 0 THEN
    // New command detected
    VO_Is_New_Command := TRUE;
    VO_Processed_ID := VI_Command_ID;
    
    // Add to history
    L_Processed_History[L_History_Index] := VI_Command_ID;
    L_Processed_Times[L_History_Index] := VI_System_Time_MS;
    L_History_Index := L_History_Index + 1;
    IF L_History_Index > GVL_CONSTANTS.C_MAX_DEDUPLICATION_HISTORY-1 THEN
        L_History_Index := 0;
    END_IF;
ELSE
    // Duplicate or empty command
    VO_Is_New_Command := FALSE;
    VO_Processed_ID := 0;
END_IF;
          
END_FUNCTION_BLOCK

FUNCTION_BLOCK FB_Water_Isolation_Authority_Arbitrator
  VAR_INPUT
    VI_Enable : BOOL;
    VI_System_Time_MS : UDINT;
  END_VAR
  VAR
    L_i : INT;
    L_Runtime : ST_Water_Isolation_Runtime_State;
    L_Traversal : ST_Water_Graph_Traversal_State;
    L_Authority : ST_Water_Isolation_Authority_State;
    L_Any_Selective : BOOL;
    L_Any_Global : BOOL;
    L_Any_Denied : BOOL;
  END_VAR

            IF NOT VI_Enable THEN
    GVL_Water_Isolation_Authority.G_Authority_Valid := FALSE;
    RETURN;
END_IF;

FOR L_i := 1 TO GVL_CONSTANTS.C_MAX_FLOOD_SENSORS DO

    L_Runtime := GVL_Water_Isolation_Runtime.G_Isolation_Runtime_State[L_i];
    L_Traversal := GVL_Water_Orchestration.G_Traversal_State[L_i];

    L_Authority := (Decision_Valid := TRUE);
    L_Authority.Decision_System_Time_MS := VI_System_Time_MS;

    L_Authority.Isolation_Requested := L_Runtime.Isolation_Requested;
    L_Authority.Selective_Candidate := L_Runtime.Selective_Isolation_Requested;
    L_Authority.Global_Fallback_Candidate := L_Runtime.Global_Isolation_Requested;

    L_Authority.Hydraulic_Zone_Id := L_Runtime.Hydraulic_Zone_Id;
    L_Authority.Isolation_Group_Id := L_Runtime.Isolation_Group_Id;
    L_Authority.Valve_Group_Id := L_Runtime.Valve_Group_Id;

    // Orchestration-derived authority.
    L_Authority.Mapping_Valid := L_Traversal.Traversal_Valid;

    L_Authority.Deterministic_Target_Valid :=
        (L_Runtime.Valve_Group_Id <> 0)
        AND NOT L_Traversal.Traversal_Conflict
        AND NOT L_Traversal.Traversal_Ambiguous;

    L_Authority.Safety_Context_Allows_Selective :=
        NOT GVL_INTENT_SAFETY.I_Water_Main_Close_Required;

    IF NOT L_Authority.Isolation_Requested THEN

        L_Authority.Decision_Code := 0;
        L_Authority.Decision_Text := 'No authority required';

    ELSIF NOT L_Authority.Mapping_Valid
       OR NOT L_Authority.Deterministic_Target_Valid
       OR NOT L_Authority.Safety_Context_Allows_Selective THEN

        L_Authority.Global_Fallback_Required := TRUE;
        L_Authority.Authority_Denied := TRUE;

        L_Authority.Decision_Code := 2;
        L_Authority.Decision_Text := 'Global fallback authority active';

    ELSE

        L_Authority.Selective_Authority_Allowed := TRUE;

        L_Authority.Decision_Code := 10;
        L_Authority.Decision_Text := 'Selective authority granted';

    END_IF;

    GVL_Water_Isolation_Authority.G_Authority_State[L_i] :=
        L_Authority;

    L_Any_Selective :=
        L_Any_Selective
        OR L_Authority.Selective_Authority_Allowed;

    L_Any_Global :=
        L_Any_Global
        OR L_Authority.Global_Fallback_Required;

    L_Any_Denied :=
        L_Any_Denied
        OR L_Authority.Authority_Denied;

END_FOR;

GVL_Water_Isolation_Authority.G_Any_Selective_Authority_Allowed :=
    L_Any_Selective;

GVL_Water_Isolation_Authority.G_Any_Global_Fallback_Required :=
    L_Any_Global;

GVL_Water_Isolation_Authority.G_Any_Authority_Denied :=
    L_Any_Denied;

GVL_Water_Isolation_Authority.G_Authority_Valid := TRUE;
GVL_Water_Isolation_Authority.G_Last_Update_MS := VI_System_Time_MS;

IF L_Any_Global THEN
    GVL_Water_Isolation_Authority.G_Status_Code := 2;
    GVL_Water_Isolation_Authority.G_Status_Text :=
        'Global fallback authority active';
ELSIF L_Any_Selective THEN
    GVL_Water_Isolation_Authority.G_Status_Code := 1;
    GVL_Water_Isolation_Authority.G_Status_Text :=
        'Selective orchestration authority active';
ELSE
    GVL_Water_Isolation_Authority.G_Status_Code := 0;
    GVL_Water_Isolation_Authority.G_Status_Text :=
        'Authority arbitration healthy';
END_IF;
          
END_FUNCTION_BLOCK

FUNCTION_BLOCK FB_Simulation_Manager
  VAR_INPUT
    VI_System_Time_MS : UDINT;
    VI_IsActivePLC : BOOL;
    VI_Scenario : E_SCENARIO_TYPE;
    VI_Config : ST_Scenario_Config;
  END_VAR
  VAR_OUTPUT
    VO_Sim_Lights : ARRAY[1..32] OF BOOL;
    VO_Sim_Active : BOOL;
    VO_Sim_Water_Leak : ARRAY[1..GVL_CONSTANTS.C_MAX_FLOOD_SENSORS] OF BOOL;
    VO_Sim_Gas_Leak : ARRAY[1..GVL_CONSTANTS.C_MAX_METHANE_SENSORS] OF REAL;
  END_VAR
  VAR
    L_Last_Toggle : UDINT;
    L_i : INT;
    L_Slot : UDINT;
  END_VAR

            IF (NOT VI_IsActivePLC) THEN
    VO_Sim_Active := FALSE;
    FOR L_i := 1 TO 32 DO
        VO_Sim_Lights[L_i] := FALSE;
    END_FOR;
    FOR L_i := 1 TO GVL_CONSTANTS.C_MAX_FLOOD_SENSORS DO
        VO_Sim_Water_Leak[L_i] := FALSE;
    END_FOR;
    FOR L_i := 1 TO GVL_CONSTANTS.C_MAX_METHANE_SENSORS DO
        VO_Sim_Gas_Leak[L_i] := REAL#0.0;
    END_FOR;
    RETURN;
END_IF;

IF (VI_Scenario = E_SCENARIO_TYPE.SCENARIO_AWAY) AND VI_Config.Presence_Simulation_Enabled THEN
    VO_Sim_Active := TRUE;

    IF (VI_System_Time_MS - L_Last_Toggle) >= (GVL_CONSTANTS.C_MS_IN_MINUTE * 30) THEN
        L_Last_Toggle := VI_System_Time_MS;
        L_Slot := (VI_System_Time_MS / GVL_CONSTANTS.C_MS_IN_MINUTE) MOD 32;

        FOR L_i := 1 TO 32 DO
            VO_Sim_Lights[L_i] := ((TO_UDINT(L_i) + L_Slot) MOD 5) = 0;
        END_FOR;
    END_IF;
ELSE
    VO_Sim_Active := FALSE;
    FOR L_i := 1 TO 32 DO
        VO_Sim_Lights[L_i] := FALSE;
    END_FOR;
END_IF;

FOR L_i := 1 TO GVL_CONSTANTS.C_MAX_FLOOD_SENSORS DO
    VO_Sim_Water_Leak[L_i] := FALSE;
END_FOR;
FOR L_i := 1 TO GVL_CONSTANTS.C_MAX_METHANE_SENSORS DO
    VO_Sim_Gas_Leak[L_i] := REAL#0.0;
END_FOR;

// >>> BULK_SYNC_ANCHOR: FB_Simulation_Manager <<<
          
END_FUNCTION_BLOCK

FUNCTION_BLOCK FB_Heating_Runtime_Observer
  VAR_INPUT
    VI_Enable : BOOL;
    VI_Runtime_Context : ST_Heating_Runtime_Context;
    VI_Diagnostics_Valid : BOOL;
  END_VAR
  VAR_OUTPUT
    VO_Observation : ST_Heating_Runtime_Observation;
    VO_Observer_Ready : BOOL;
    VO_Observer_Fault : BOOL;
    VO_Status_Code : UINT;
    VO_Status_Text : STRING(128);
  END_VAR

            // ==============================================================================
// Heating runtime observer
// Minimal observer-only runtime attachment.
// Read-only.
// Governance-locked.
// Finalized-state observation only.
// ==============================================================================



// ======================================================
// DEFAULTS
// ======================================================
VO_Observation.Runtime_Active := FALSE;
VO_Observation.Runtime_Ready := FALSE;
VO_Observation.Runtime_Fault := FALSE;
VO_Observation.Current_Phase := E_Heating_Runtime_Phase.HRP_DISABLED;

VO_Observation.DHW_Demand_Active := FALSE;
VO_Observation.DHW_Heating_Active := FALSE;
VO_Observation.DHW_Circulation_Active := FALSE;

VO_Observation.Heating_Demand_Active := FALSE;
VO_Observation.Heating_Runtime_Active := FALSE;
VO_Observation.Heating_Output_Active := FALSE;

VO_Observation.Cascade_Available := FALSE;
VO_Observation.Cascade_Degraded := FALSE;
VO_Observation.Cascade_Active_Boilers := 0;
VO_Observation.Cascade_Available_Boilers := 0;

VO_Observation.OpenTherm_Online := FALSE;
VO_Observation.OpenTherm_Command_Valid := FALSE;
VO_Observation.OpenTherm_Transport_Degraded := FALSE;

VO_Observation.Diagnostics_Active := FALSE;
VO_Observation.Explainability_Active := FALSE;

VO_Observation.DHW_Before_Heating_Observed := FALSE;
VO_Observation.Diagnostics_After_Publication_Observed := FALSE;
VO_Observation.Output_Projection_Last_Observed := FALSE;

VO_Observation.Runtime_Ownership_Valid := TRUE;
VO_Observation.Diagnostics_Ownership_Valid := TRUE;
VO_Observation.OpenTherm_Ownership_Valid := TRUE;
VO_Observation.Cascade_Ownership_Valid := TRUE;
VO_Observation.Safety_Ownership_Valid := TRUE;

VO_Observation.Observation_Status_Code := 0;
VO_Observation.Observation_Status_Text := 'Heating runtime observer disabled';

VO_Observer_Ready := FALSE;
VO_Observer_Fault := FALSE;
VO_Status_Code := 0;
VO_Status_Text := 'Heating runtime observer disabled';

IF NOT VI_Enable THEN
    RETURN;
END_IF;

// ======================================================
// FINALIZED-STATE OBSERVATION ONLY
// ======================================================
VO_Observation.Runtime_Active := VI_Runtime_Context.Runtime_Enabled;
VO_Observation.Runtime_Ready := VI_Runtime_Context.Runtime_Ready;
VO_Observation.Runtime_Fault := VI_Runtime_Context.Runtime_Fault;
VO_Observation.Current_Phase := VI_Runtime_Context.Current_Phase;

VO_Observation.Diagnostics_Active := VI_Diagnostics_Valid;
VO_Observation.Explainability_Active := VI_Runtime_Context.Explainability_Isolation_Valid;

VO_Observation.DHW_Before_Heating_Observed :=
    VI_Runtime_Context.DHW_Before_Heating_Valid;

VO_Observation.Diagnostics_After_Publication_Observed :=
    VI_Runtime_Context.State_Publication_Before_Diagnostics_Valid;

VO_Observation.Output_Projection_Last_Observed :=
    VI_Runtime_Context.Output_Projection_Last_Valid;

VO_Observation.Runtime_Ownership_Valid := TRUE;
VO_Observation.Diagnostics_Ownership_Valid :=
    VI_Runtime_Context.Diagnostics_Isolation_Valid;

VO_Observation.OpenTherm_Ownership_Valid :=
    VI_Runtime_Context.OpenTherm_Ownership_Valid;

VO_Observation.Cascade_Ownership_Valid :=
    VI_Runtime_Context.Cascade_Ownership_Valid;

VO_Observation.Safety_Ownership_Valid :=
    VI_Runtime_Context.Safety_Isolation_Valid;

// These domain-specific runtime values remain intentionally FALSE/0 here.
// They must be populated only by finalized publication contracts, not by internal runtime scans.
VO_Observation.DHW_Demand_Active := FALSE;
VO_Observation.DHW_Heating_Active := FALSE;
VO_Observation.DHW_Circulation_Active := FALSE;
VO_Observation.Heating_Demand_Active := FALSE;
VO_Observation.Heating_Runtime_Active := FALSE;
VO_Observation.Heating_Output_Active := FALSE;
VO_Observation.Cascade_Available := FALSE;
VO_Observation.Cascade_Degraded := FALSE;
VO_Observation.Cascade_Active_Boilers := 0;
VO_Observation.Cascade_Available_Boilers := 0;
VO_Observation.OpenTherm_Online := FALSE;
VO_Observation.OpenTherm_Command_Valid := FALSE;
VO_Observation.OpenTherm_Transport_Degraded := FALSE;

// ======================================================
// STATUS
// ======================================================
IF VI_Runtime_Context.Runtime_Fault THEN
    VO_Observation.Observation_Status_Code := 900;
    VO_Observation.Observation_Status_Text := 'Heating runtime observer detected runtime fault';

ELSIF NOT VI_Diagnostics_Valid THEN
    VO_Observation.Observation_Status_Code := 200;
    VO_Observation.Observation_Status_Text := 'Heating runtime diagnostics publication invalid';

ELSE
    VO_Observation.Observation_Status_Code := 1;
    VO_Observation.Observation_Status_Text := 'Heating runtime observer nominal';
END_IF;

VO_Observer_Ready := TRUE;
VO_Observer_Fault := FALSE;

VO_Status_Code := VO_Observation.Observation_Status_Code;
VO_Status_Text := VO_Observation.Observation_Status_Text;

// >>> BULK_SYNC_ANCHOR: FB_Heating_Runtime_Observer <<<
          
END_FUNCTION_BLOCK

FUNCTION_BLOCK FB_Heating_Runtime_OT_Cascade_Correlator
  VAR_INPUT
    VI_Enable : BOOL;
    VI_Cascade_Degraded : BOOL;
    VI_OT_Degraded : BOOL;
    VI_OT_Command_Valid : BOOL;
    VI_Boiler_Count : UINT;
  END_VAR
  VAR_OUTPUT
    VO_Correlation_Detected : BOOL;
    VO_Status_Code : UINT;
    VO_Status_Text : STRING(128);
  END_VAR

            // ==============================================================================
// Heating runtime OT and cascade correlator
// Read-only degradation correlation layer.
// ==============================================================================



VO_Correlation_Detected := FALSE;
VO_Status_Code := 0;
VO_Status_Text := 'Heating OT/cascade correlator disabled';

IF NOT VI_Enable THEN
    RETURN;
END_IF;

VO_Correlation_Detected :=
    VI_Cascade_Degraded OR
    VI_OT_Degraded OR
    NOT VI_OT_Command_Valid OR
    (VI_Boiler_Count = 0);

IF VO_Correlation_Detected THEN
    VO_Status_Code := 200;
    VO_Status_Text := 'Heating OT/cascade degradation correlated';
ELSE
    VO_Status_Code := 1;
    VO_Status_Text := 'Heating OT/cascade nominal';
END_IF;

// >>> BULK_SYNC_ANCHOR: FB_Heating_Runtime_OT_Cascade_Correlator <<<
          
END_FUNCTION_BLOCK

FUNCTION_BLOCK FB_System_Gateway_Intent
  VAR_INPUT
    VI_System_Time_MS : UDINT;
    VI_IsActivePLC : BOOL;
    VI_Gateway_Writes_Allowed : BOOL;
  END_VAR
  VAR_IN_OUT
    VIO_FloorHeating_Temps : ARRAY[1..GVL_CONSTANTS.C_MAX_HEATING_CIRCUITS] OF REAL;
    VIO_Zone_Valve_States : ARRAY[1..GVL_CONSTANTS.C_MAX_HEATING_CIRCUITS] OF BOOL;
    VIO_Lighting_Base_Levels : ARRAY[1..GVL_CONSTANTS.C_MAX_LIGHT_ZONES] OF BYTE;
    VIO_Scenario_Req_Gateway : E_SCENARIO_TYPE;
  END_VAR
  VAR
    fbGateway : FB_Gateway_Interface;
    L_Gateway_Flood_Alarm_Active : BOOL;
    L_Gateway_Gas_Alarm_Active : BOOL;
    L_Gateway_Fire_Alarm_Active : BOOL;
  END_VAR

            // Gateway telemetry must expose authoritative safety truth and latches,
// not stale alarm projection fields.
L_Gateway_Flood_Alarm_Active := GVL_HEALTH_BRIDGE.G_Leak_Detected OR GVL_STATE.G_Safety_Leak_Latched;
L_Gateway_Gas_Alarm_Active := GVL_HEALTH_BRIDGE.G_Gas_Detected OR GVL_HEALTH_BRIDGE.G_CO_Alarm_Level OR GVL_STATE.G_Safety_Gas_Latched;
L_Gateway_Fire_Alarm_Active := GVL_HEALTH_BRIDGE.G_Smoke_Detected OR GVL_STATE.G_Safety_Smoke_Latched;

